LIN {X 0,Y 213.774,Z 837.959,A -85,B 0,C 180,E1 9874.512,E2 9874.512} C_VEL
LIN {X 0,Y 216.495,Z 837.046,A -85,B 0,C 180,E1 9873.088,E2 9873.088} C_VEL
LIN {X 0,Y 220.034,Z 835.344,A -85,B 0,C 180,E1 9871.796,E2 9871.796} C_VEL
LIN {X 0,Y 223.983,Z 833.719,A -85,B 0,C 180,E1 9870.296,E2 9870.296} C_VEL
LIN {X 0,Y 226.594,Z 832.46,A -85,B 0,C 180,E1 9869.505,E2 9869.505} C_VEL
LIN {X 0,Y 231.577,Z 830.349,A -85,B 0,C 180,E1 9867.921,E2 9867.921} C_VEL
LIN {X 0,Y 234.959,Z 828.778,A -85,B 0,C 180,E1 9866.995,E2 9866.995} C_VEL
LIN {X 0,Y 241.29,Z 825.829,A -85,B 0,C 180,E1 9865.408,E2 9865.408} C_VEL
LIN {X 0,Y 250.192,Z 821.605,A -85,B 0,C 180,E1 9863.446,E2 9863.446} C_VEL
LIN {X 0,Y 261.296,Z 816.099,A -85,B 0,C 180,E1 9861.41,E2 9861.41} C_VEL
LIN {X 0,Y 266.545,Z 813.328,A -85,B 0,C 180,E1 9860.587,E2 9860.587} C_VEL
LIN {X 0,Y 257.171,Z 829.628,A -85,B 0,C 180,E1 9857.623,E2 9857.623} C_VEL
LIN {X 0,Y 247.802,Z 844.317,A -85,B 0,C 180,E1 9854.272,E2 9854.272} C_VEL
LIN {X 0,Y 238.695,Z 857.461,A -85,B 0,C 180,E1 9850.488,E2 9850.488} C_VEL
LIN {X 0,Y 230.087,Z 869.099,A -85,B 0,C 180,E1 9846.229,E2 9846.229} C_VEL
LIN {X 0,Y 222.258,Z 879.206,A -85,B 0,C 180,E1 9841.457,E2 9841.457} C_VEL
LIN {X 0,Y 215.768,Z 887.387,A -85,B 0,C 180,E1 9836.415,E2 9836.415} C_VEL
LIN {X 0,Y 210.469,Z 894.092,A -85,B 0,C 180,E1 9830.874,E2 9830.874} C_VEL
LIN {X 0,Y 206.702,Z 899.028,A -85,B 0,C 180,E1 9825.143,E2 9825.143} C_VEL
LIN {X 0,Y 204.391,Z 902.303,A -85,B 0,C 180,E1 9819.291,E2 9819.291} C_VEL
LIN {X 0,Y 203.309,Z 903.961,A -85,B 0,C 180,E1 9813.384,E2 9813.384} C_VEL
LIN {X 0,Y 203.212,Z 904.09,A -85,B 0,C 180,E1 9807.744,E2 9807.744} C_VEL
LIN {X 0,Y 204.008,Z 902.842,A -85,B 0,C 180,E1 9802.112,E2 9802.112} C_VEL
LIN {X 0,Y 206.112,Z 899.833,A -85,B 0,C 180,E1 9795.963,E2 9795.963} C_VEL
LIN {X 0,Y 209.786,Z 895.013,A -85,B 0,C 180,E1 9789.93,E2 9789.93} C_VEL
LIN {X 0,Y 214.836,Z 888.617,A -85,B 0,C 180,E1 9784.352,E2 9784.352} C_VEL
LIN {X 0,Y 221.454,Z 880.322,A -85,B 0,C 180,E1 9779.021,E2 9779.021} C_VEL
LIN {X 0,Y 229.143,Z 870.475,A -85,B 0,C 180,E1 9774.217,E2 9774.217} C_VEL
LIN {X 0,Y 237.624,Z 859.12,A -85,B 0,C 180,E1 9769.924,E2 9769.924} C_VEL
LIN {X 0,Y 246.624,Z 846.271,A -85,B 0,C 180,E1 9766.109,E2 9766.109} C_VEL
LIN {X 0,Y 255.338,Z 832.826,A -85,B 0,C 180,E1 9762.922,E2 9762.922} C_VEL
LIN {X 0,Y 264.272,Z 817.707,A -85,B 0,C 180,E1 9760.032,E2 9760.032} C_VEL
LIN {X 0,Y 272.923,Z 801.409,A -85,B 0,C 180,E1 9757.517,E2 9757.517} C_VEL
LIN {X 0,Y 281.204,Z 783.726,A -85,B 0,C 180,E1 9755.309,E2 9755.309} C_VEL
LIN {X 0,Y 288.732,Z 765.064,A -85,B 0,C 180,E1 9753.427,E2 9753.427} C_VEL
LIN {X 0,Y 295.016,Z 746.597,A -85,B 0,C 180,E1 9751.92,E2 9751.92} C_VEL
LIN {X 0,Y 300.676,Z 726.186,A -85,B 0,C 180,E1 9750.584,E2 9750.584} C_VEL
LIN {X 0,Y 305.859,Z 701.959,A -85,B 0,C 180,E1 9749.35,E2 9749.35} C_VEL
LIN {X 0,Y 313.548,Z 662.516,A -85,B 0,C 180,E1 9747.755,E2 9747.755} C_VEL
LIN {X 0,Y 320.97,Z 622.102,A -85,B 0,C 180,E1 9746.524,E2 9746.524} C_VEL
LIN {X 0,Y 328.272,Z 576.098,A -85,B 0,C 180,E1 9745.404,E2 9745.404} C_VEL
LIN {X 0,Y 333.972,Z 529.706,A -85,B 0,C 180,E1 9744.467,E2 9744.467} C_VEL
LIN {X 0,Y 340.15,Z 466.539,A -85,B 0,C 180,E1 9743.356,E2 9743.356} C_VEL
LIN {X 0,Y 344.086,Z 450.132,A -85,B 0,C 180,E1 9742.901,E2 9742.901} C_VEL
LIN {X 0,Y 341.351,Z 438.925,A -85,B 0,C 180,E1 9739.82,E2 9739.82} C_VEL
LIN {X 0,Y 340.469,Z 435.442,A -85,B 0,C 180,E1 9738.706,E2 9738.706} C_VEL
LIN {X 0,Y 339.282,Z 432.899,A -85,B 0,C 180,E1 9737.488,E2 9737.488} C_VEL
LIN {X 0,Y 336.733,Z 431.213,A -85,B 0,C 180,E1 9735.367,E2 9735.367} C_VEL
LIN {X 0,Y 334.628,Z 429.482,A -85,B 0,C 180,E1 9733.301,E2 9733.301} C_VEL
LIN {X 0,Y 334.307,Z 428.715,A -85,B 0,C 180,E1 9732.841,E2 9732.841} C_VEL
LIN {X 0,Y 332.924,Z 422.507,A -85,B 0,C 180,E1 9729.421,E2 9729.421} C_VEL
LIN {X 0,Y 332.056,Z 418.778,A -85,B 0,C 180,E1 9726.571,E2 9726.571} C_VEL
LIN {X 0,Y 331.825,Z 415.306,A -85,B 0,C 180,E1 9722.936,E2 9722.936} C_VEL
LIN {X 0,Y 332.528,Z 414.439,A -85,B 0,C 180,E1 9717.932,E2 9717.932} C_VEL
LIN {X 0,Y 333.593,Z 415.275,A -85,B 0,C 180,E1 9715.186,E2 9715.186} C_VEL
LIN {X 0,Y 334.377,Z 429.017,A -85,B 0,C 180,E1 9710.621,E2 9710.621} C_VEL
LIN {X 0,Y 337.146,Z 447.925,A -85,B 0,C 180,E1 9705.443,E2 9705.443} C_VEL
LIN {X 0,Y 337.566,Z 450.515,A -85,B 0,C 180,E1 9704.861,E2 9704.861} C_VEL
LIN {X 0,Y 319.756,Z 552.113,A -85,B 0,C 180,E1 9702.274,E2 9702.274} C_VEL
LIN {X 0,Y 313.651,Z 616.805,A -85,B 0,C 180,E1 9700.912,E2 9700.912} C_VEL
LIN {X 0,Y 308.573,Z 653.152,A -85,B 0,C 180,E1 9700.066,E2 9700.066} C_VEL
LIN {X 0,Y 302.296,Z 687.872,A -85,B 0,C 180,E1 9699.032,E2 9699.032} C_VEL
LIN {X 0,Y 294.882,Z 721.646,A -85,B 0,C 180,E1 9697.789,E2 9697.789} C_VEL
LIN {X 0,Y 287.35,Z 751.978,A -85,B 0,C 180,E1 9696.384,E2 9696.384} C_VEL
LIN {X 0,Y 278.355,Z 784.046,A -85,B 0,C 180,E1 9694.465,E2 9694.465} C_VEL
LIN {X 0,Y 272.028,Z 802.983,A -85,B 0,C 180,E1 9693.044,E2 9693.044} C_VEL
LIN {X 0,Y 264.192,Z 822.641,A -85,B 0,C 180,E1 9691.182,E2 9691.182} C_VEL
LIN {X 0,Y 255.628,Z 841.24,A -85,B 0,C 180,E1 9688.939,E2 9688.939} C_VEL
LIN {X 0,Y 246.829,Z 858.228,A -85,B 0,C 180,E1 9686.353,E2 9686.353} C_VEL
LIN {X 0,Y 237.72,Z 874.11,A -85,B 0,C 180,E1 9683.325,E2 9683.325} C_VEL
LIN {X 0,Y 228.326,Z 889.305,A -85,B 0,C 180,E1 9679.639,E2 9679.639} C_VEL
LIN {X 0,Y 219.526,Z 902.891,A -85,B 0,C 180,E1 9675.457,E2 9675.457} C_VEL
LIN {X 0,Y 211.133,Z 915.618,A -85,B 0,C 180,E1 9670.452,E2 9670.452} C_VEL
LIN {X 0,Y 204.191,Z 926.472,A -85,B 0,C 180,E1 9664.955,E2 9664.955} C_VEL
LIN {X 0,Y 198.818,Z 935.674,A -85,B 0,C 180,E1 9658.868,E2 9658.868} C_VEL
LIN {X 0,Y 195.438,Z 942.931,A -85,B 0,C 180,E1 9652.564,E2 9652.564} C_VEL
LIN {X 0,Y 193.909,Z 948.606,A -85,B 0,C 180,E1 9645.86,E2 9645.86} C_VEL
LIN {X 0,Y 193.96,Z 952.104,A -85,B 0,C 180,E1 9639.795,E2 9639.795} C_VEL
LIN {X 0,Y 194.718,Z 953.916,A -85,B 0,C 180,E1 9634.417,E2 9634.417} C_VEL
LIN {X 0,Y 195.109,Z 954.446,A -85,B 0,C 180,E1 9630,E2 9630} C_VEL
LIN {X 0,Y 194.783,Z 953.918,A -85,B 0,C 180,E1 9625.584,E2 9625.584} C_VEL
LIN {X 0,Y 194.115,Z 952.266,A -85,B 0,C 180,E1 9619.913,E2 9619.913} C_VEL
LIN {X 0,Y 193.988,Z 951.89,A -85,B 0,C 180,E1 9613.223,E2 9613.223} C_VEL
LIN {X 0,Y 196.359,Z 949.933,A -85,B 0,C 180,E1 9605.319,E2 9605.319} C_VEL
LIN {X 0,Y 203.821,Z 945.545,A -85,B 0,C 180,E1 9595.996,E2 9595.996} C_VEL
LIN {X 0,Y 216.327,Z 939.485,A -85,B 0,C 180,E1 9587.559,E2 9587.559} C_VEL
LIN {X 0,Y 235.213,Z 931.168,A -85,B 0,C 180,E1 9579.697,E2 9579.697} C_VEL
LIN {X 0,Y 245.482,Z 926.927,A -85,B 0,C 180,E1 9576.57,E2 9576.57} C_VEL
LIN {X 0,Y 230.871,Z 927.562,A -85,B 0,C 180,E1 9571.896,E2 9571.896} C_VEL
LIN {X 0,Y 218.657,Z 926.56,A -85,B 0,C 180,E1 9566.625,E2 9566.625} C_VEL
LIN {X 0,Y 209.607,Z 924.018,A -85,B 0,C 180,E1 9561.257,E2 9561.257} C_VEL
LIN {X 0,Y 202.738,Z 919.727,A -85,B 0,C 180,E1 9555.446,E2 9555.446} C_VEL
LIN {X 0,Y 198.06,Z 913.469,A -85,B 0,C 180,E1 9549.297,E2 9549.297} C_VEL
LIN {X 0,Y 195.581,Z 905.888,A -85,B 0,C 180,E1 9543.517,E2 9543.517} C_VEL
LIN {X 0,Y 194.576,Z 897.367,A -85,B 0,C 180,E1 9538.233,E2 9538.233} C_VEL
LIN {X 0,Y 194.552,Z 887.031,A -85,B 0,C 180,E1 9532.915,E2 9532.915} C_VEL
LIN {X 0,Y 195.453,Z 874.895,A -85,B 0,C 180,E1 9527.718,E2 9527.718} C_VEL
LIN {X 0,Y 197.218,Z 861.476,A -85,B 0,C 180,E1 9522.899,E2 9522.899} C_VEL
LIN {X 0,Y 199.677,Z 847.469,A -85,B 0,C 180,E1 9518.558,E2 9518.558} C_VEL
LIN {X 0,Y 201.324,Z 847.012,A -85,B 0,C 180,E1 9517.208,E2 9517.208} C_VEL
LIN {X 0,Y 204.017,Z 845.607,A -85,B 0,C 180,E1 9515.997,E2 9515.997} C_VEL
LIN {X 0,Y 206.542,Z 844.763,A -85,B 0,C 180,E1 9514.478,E2 9514.478} C_VEL
LIN {X 0,Y 209.844,Z 843.247,A -85,B 0,C 180,E1 9513.085,E2 9513.085} C_VEL
LIN {X 0,Y 213.572,Z 841.761,A -85,B 0,C 180,E1 9511.475,E2 9511.475} C_VEL
LIN {X 0,Y 215.992,Z 840.669,A -85,B 0,C 180,E1 9510.613,E2 9510.613} C_VEL
LIN {X 0,Y 220.769,Z 838.719,A -85,B 0,C 180,E1 9508.914,E2 9508.914} C_VEL
LIN {X 0,Y 229.354,Z 835.015,A -85,B 0,C 180,E1 9506.376,E2 9506.376} C_VEL
LIN {X 0,Y 237.845,Z 831.343,A -85,B 0,C 180,E1 9504.243,E2 9504.243} C_VEL
LIN {X 0,Y 247.768,Z 826.829,A -85,B 0,C 180,E1 9502.163,E2 9502.163} C_VEL
LIN {X 0,Y 256.771,Z 822.752,A -85,B 0,C 180,E1 9500.496,E2 9500.496} C_VEL
LIN {X 0,Y 247.225,Z 837.953,A -85,B 0,C 180,E1 9497.4,E2 9497.4} C_VEL
LIN {X 0,Y 237.316,Z 852.257,A -85,B 0,C 180,E1 9493.709,E2 9493.709} C_VEL
LIN {X 0,Y 228.297,Z 864.319,A -85,B 0,C 180,E1 9489.751,E2 9489.751} C_VEL
LIN {X 0,Y 219.841,Z 874.97,A -85,B 0,C 180,E1 9485.284,E2 9485.284} C_VEL
LIN {X 0,Y 212.23,Z 884.171,A -85,B 0,C 180,E1 9480.273,E2 9480.273} C_VEL
LIN {X 0,Y 205.696,Z 891.933,A -85,B 0,C 180,E1 9474.631,E2 9474.631} C_VEL
LIN {X 0,Y 200.728,Z 897.907,A -85,B 0,C 180,E1 9468.591,E2 9468.591} C_VEL
LIN {X 0,Y 197.535,Z 901.951,A -85,B 0,C 180,E1 9462.572,E2 9462.572} C_VEL
LIN {X 0,Y 195.79,Z 904.377,A -85,B 0,C 180,E1 9456.451,E2 9456.451} C_VEL
LIN {X 0,Y 195.217,Z 905.198,A -85,B 0,C 180,E1 9450.587,E2 9450.587} C_VEL
LIN {X 0,Y 195.576,Z 904.642,A -85,B 0,C 180,E1 9444.72,E2 9444.72} C_VEL
LIN {X 0,Y 197.067,Z 902.567,A -85,B 0,C 180,E1 9438.587,E2 9438.587} C_VEL
LIN {X 0,Y 200.126,Z 898.677,A -85,B 0,C 180,E1 9432.256,E2 9432.256} C_VEL
LIN {X 0,Y 204.905,Z 892.926,A -85,B 0,C 180,E1 9426.108,E2 9426.108} C_VEL
LIN {X 0,Y 211.121,Z 885.568,A -85,B 0,C 180,E1 9420.492,E2 9420.492} C_VEL
LIN {X 0,Y 218.51,Z 876.704,A -85,B 0,C 180,E1 9415.43,E2 9415.43} C_VEL
LIN {X 0,Y 226.846,Z 866.319,A -85,B 0,C 180,E1 9410.876,E2 9410.876} C_VEL
LIN {X 0,Y 235.805,Z 854.497,A -85,B 0,C 180,E1 9406.831,E2 9406.831} C_VEL
LIN {X 0,Y 245.117,Z 841.277,A -85,B 0,C 180,E1 9403.26,E2 9403.26} C_VEL
LIN {X 0,Y 254.736,Z 826.348,A -85,B 0,C 180,E1 9400.056,E2 9400.056} C_VEL
LIN {X 0,Y 264.011,Z 810.344,A -85,B 0,C 180,E1 9397.313,E2 9397.313} C_VEL
LIN {X 0,Y 272.725,Z 793.383,A -85,B 0,C 180,E1 9394.974,E2 9394.974} C_VEL
LIN {X 0,Y 280.716,Z 775.526,A -85,B 0,C 180,E1 9392.983,E2 9392.983} C_VEL
LIN {X 0,Y 287.85,Z 756.807,A -85,B 0,C 180,E1 9391.294,E2 9391.294} C_VEL
LIN {X 0,Y 294.047,Z 737.187,A -85,B 0,C 180,E1 9389.875,E2 9389.875} C_VEL
LIN {X 0,Y 299.024,Z 717.296,A -85,B 0,C 180,E1 9388.727,E2 9388.727} C_VEL
LIN {X 0,Y 306.803,Z 679.572,A -85,B 0,C 180,E1 9387.046,E2 9387.046} C_VEL
LIN {X 0,Y 314.484,Z 640.094,A -85,B 0,C 180,E1 9385.7,E2 9385.7} C_VEL
LIN {X 0,Y 322.291,Z 594.861,A -85,B 0,C 180,E1 9384.537,E2 9384.537} C_VEL
LIN {X 0,Y 328.535,Z 550.082,A -85,B 0,C 180,E1 9383.578,E2 9383.578} C_VEL
LIN {X 0,Y 334.258,Z 494.763,A -85,B 0,C 180,E1 9382.586,E2 9382.586} C_VEL
LIN {X 0,Y 336.896,Z 469.242,A -85,B 0,C 180,E1 9382.144,E2 9382.144} C_VEL
LIN {X 0,Y 340.426,Z 454.288,A -85,B 0,C 180,E1 9381.721,E2 9381.721} C_VEL
LIN {X 0,Y 338.052,Z 443.9,A -85,B 0,C 180,E1 9378.719,E2 9378.719} C_VEL
LIN {X 0,Y 335.855,Z 434.787,A -85,B 0,C 180,E1 9375.498,E2 9375.498} C_VEL
LIN {X 0,Y 334.307,Z 428.715,A -85,B 0,C 180,E1 9372.841,E2 9372.841} C_VEL
LIN {X 0,Y 333.429,Z 427.235,A -85,B 0,C 180,E1 9371.542,E2 9371.542} C_VEL
LIN {X 0,Y 331.509,Z 427.281,A -85,B 0,C 180,E1 9369.153,E2 9369.153} C_VEL
LIN {X 0,Y 330.247,Z 427.072,A -85,B 0,C 180,E1 9367.119,E2 9367.119} C_VEL
LIN {X 0,Y 330.126,Z 426.75,A -85,B 0,C 180,E1 9366.734,E2 9366.734} C_VEL
LIN {X 0,Y 329.901,Z 423.004,A -85,B 0,C 180,E1 9362.606,E2 9362.606} C_VEL
LIN {X 0,Y 330.781,Z 422.255,A -85,B 0,C 180,E1 9357.748,E2 9357.748} C_VEL
LIN {X 0,Y 331.614,Z 422.963,A -85,B 0,C 180,E1 9355.504,E2 9355.504} C_VEL
LIN {X 0,Y 332.18,Z 436.644,A -85,B 0,C 180,E1 9350.995,E2 9350.995} C_VEL
LIN {X 0,Y 334.634,Z 454.529,A -85,B 0,C 180,E1 9346.085,E2 9346.085} C_VEL
LIN {X 0,Y 317.576,Z 549.187,A -85,B 0,C 180,E1 9343.709,E2 9343.709} C_VEL
LIN {X 0,Y 311.251,Z 614.325,A -85,B 0,C 180,E1 9342.345,E2 9342.345} C_VEL
LIN {X 0,Y 305.933,Z 651.501,A -85,B 0,C 180,E1 9341.503,E2 9341.503} C_VEL
LIN {X 0,Y 299.223,Z 687.667,A -85,B 0,C 180,E1 9340.448,E2 9340.448} C_VEL
LIN {X 0,Y 291.638,Z 721.28,A -85,B 0,C 180,E1 9339.23,E2 9339.23} C_VEL
LIN {X 0,Y 283.713,Z 752.096,A -85,B 0,C 180,E1 9337.821,E2 9337.821} C_VEL
LIN {X 0,Y 275.126,Z 782.04,A -85,B 0,C 180,E1 9336.064,E2 9336.064} C_VEL
LIN {X 0,Y 268.417,Z 801.547,A -85,B 0,C 180,E1 9334.634,E2 9334.634} C_VEL
LIN {X 0,Y 260.644,Z 820.526,A -85,B 0,C 180,E1 9332.874,E2 9332.874} C_VEL
LIN {X 0,Y 252.122,Z 838.586,A -85,B 0,C 180,E1 9330.75,E2 9330.75} C_VEL
LIN {X 0,Y 243.257,Z 855.197,A -85,B 0,C 180,E1 9328.305,E2 9328.305} C_VEL
LIN {X 0,Y 233.594,Z 871.554,A -85,B 0,C 180,E1 9325.27,E2 9325.27} C_VEL
LIN {X 0,Y 224.091,Z 886.437,A -85,B 0,C 180,E1 9321.749,E2 9321.749} C_VEL
LIN {X 0,Y 214.948,Z 899.902,A -85,B 0,C 180,E1 9317.7,E2 9317.7} C_VEL
LIN {X 0,Y 206.322,Z 912.249,A -85,B 0,C 180,E1 9312.963,E2 9312.963} C_VEL
LIN {X 0,Y 198.346,Z 923.808,A -85,B 0,C 180,E1 9307.224,E2 9307.224} C_VEL
LIN {X 0,Y 192.471,Z 932.966,A -85,B 0,C 180,E1 9301.299,E2 9301.299} C_VEL
LIN {X 0,Y 188.332,Z 940.658,A -85,B 0,C 180,E1 9294.787,E2 9294.787} C_VEL
LIN {X 0,Y 186.215,Z 946.456,A -85,B 0,C 180,E1 9288.118,E2 9288.118} C_VEL
LIN {X 0,Y 185.881,Z 950.495,A -85,B 0,C 180,E1 9281.48,E2 9281.48} C_VEL
LIN {X 0,Y 186.572,Z 952.702,A -85,B 0,C 180,E1 9275.536,E2 9275.536} C_VEL
LIN {X 0,Y 187.122,Z 953.372,A -85,B 0,C 180,E1 9271.225,E2 9271.225} C_VEL
LIN {X 0,Y 187.016,Z 953.251,A -85,B 0,C 180,E1 9267.242,E2 9267.242} C_VEL
LIN {X 0,Y 186.372,Z 951.942,A -85,B 0,C 180,E1 9261.981,E2 9261.981} C_VEL
LIN {X 0,Y 186.121,Z 950.581,A -85,B 0,C 180,E1 9258.22,E2 9258.22} C_VEL
LIN {X 0,Y 186.54,Z 950.022,A -85,B 0,C 180,E1 9250.589,E2 9250.589} C_VEL
LIN {X 0,Y 190.211,Z 947.854,A -85,B 0,C 180,E1 9242.105,E2 9242.105} C_VEL
LIN {X 0,Y 200.211,Z 943.1,A -85,B 0,C 180,E1 9232.1,E2 9232.1} C_VEL
LIN {X 0,Y 215.395,Z 936.848,A -85,B 0,C 180,E1 9223.6,E2 9223.6} C_VEL
LIN {X 0,Y 235.218,Z 929.227,A -85,B 0,C 180,E1 9216.522,E2 9216.522} C_VEL
LIN {X 0,Y 220.878,Z 928.989,A -85,B 0,C 180,E1 9211.676,E2 9211.676} C_VEL
LIN {X 0,Y 208.835,Z 927.095,A -85,B 0,C 180,E1 9206.135,E2 9206.135} C_VEL
LIN {X 0,Y 200.03,Z 923.715,A -85,B 0,C 180,E1 9200.482,E2 9200.482} C_VEL
LIN {X 0,Y 193.497,Z 918.5,A -85,B 0,C 180,E1 9194.362,E2 9194.362} C_VEL
LIN {X 0,Y 189.37,Z 911.663,A -85,B 0,C 180,E1 9188.196,E2 9188.196} C_VEL
LIN {X 0,Y 187.278,Z 903.762,A -85,B 0,C 180,E1 9182.448,E2 9182.448} C_VEL
LIN {X 0,Y 186.475,Z 894.015,A -85,B 0,C 180,E1 9176.619,E2 9176.619} C_VEL
LIN {X 0,Y 186.765,Z 882.809,A -85,B 0,C 180,E1 9171.068,E2 9171.068} C_VEL
LIN {X 0,Y 187.99,Z 870.181,A -85,B 0,C 180,E1 9165.838,E2 9165.838} C_VEL
LIN {X 0,Y 190.271,Z 855.222,A -85,B 0,C 180,E1 9160.666,E2 9160.666} C_VEL
LIN {X 0,Y 190.434,Z 854.584,A -85,B 0,C 180,E1 9160.364,E2 9160.364} C_VEL
LIN {X 0,Y 191.918,Z 854.122,A -85,B 0,C 180,E1 9158.931,E2 9158.931} C_VEL
LIN {X 0,Y 194.691,Z 852.79,A -85,B 0,C 180,E1 9157.345,E2 9157.345} C_VEL
LIN {X 0,Y 197.716,Z 851.58,A -85,B 0,C 180,E1 9155.5,E2 9155.5} C_VEL
LIN {X 0,Y 199.738,Z 850.686,A -85,B 0,C 180,E1 9154.5,E2 9154.5} C_VEL
LIN {X 0,Y 203.867,Z 849.004,A -85,B 0,C 180,E1 9152.546,E2 9152.546} C_VEL
LIN {X 0,Y 210.165,Z 846.505,A -85,B 0,C 180,E1 9149.985,E2 9149.985} C_VEL
LIN {X 0,Y 217.554,Z 843.54,A -85,B 0,C 180,E1 9147.47,E2 9147.47} C_VEL
LIN {X 0,Y 225.682,Z 840.264,A -85,B 0,C 180,E1 9145.142,E2 9145.142} C_VEL
LIN {X 0,Y 235.195,Z 836.31,A -85,B 0,C 180,E1 9142.865,E2 9142.865} C_VEL
LIN {X 0,Y 246.225,Z 831.487,A -85,B 0,C 180,E1 9140.691,E2 9140.691} C_VEL
LIN {X 0,Y 247.205,Z 831.074,A -85,B 0,C 180,E1 9140.502,E2 9140.502} C_VEL
LIN {X 0,Y 237.234,Z 845.705,A -85,B 0,C 180,E1 9137.17,E2 9137.17} C_VEL
LIN {X 0,Y 227.334,Z 858.969,A -85,B 0,C 180,E1 9133.326,E2 9133.326} C_VEL
LIN {X 0,Y 217.886,Z 870.69,A -85,B 0,C 180,E1 9128.955,E2 9128.955} C_VEL
LIN {X 0,Y 209.2,Z 880.866,A -85,B 0,C 180,E1 9124.002,E2 9124.002} C_VEL
LIN {X 0,Y 201.59,Z 889.464,A -85,B 0,C 180,E1 9118.435,E2 9118.435} C_VEL
LIN {X 0,Y 195.631,Z 896.147,A -85,B 0,C 180,E1 9112.541,E2 9112.541} C_VEL
LIN {X 0,Y 191.358,Z 901.064,A -85,B 0,C 180,E1 9106.39,E2 9106.39} C_VEL
LIN {X 0,Y 188.707,Z 904.318,A -85,B 0,C 180,E1 9100.07,E2 9100.07} C_VEL
LIN {X 0,Y 187.458,Z 905.963,A -85,B 0,C 180,E1 9093.67,E2 9093.67} C_VEL
LIN {X 0,Y 187.348,Z 906.093,A -85,B 0,C 180,E1 9087.553,E2 9087.553} C_VEL
LIN {X 0,Y 188.268,Z 904.854,A -85,B 0,C 180,E1 9081.448,E2 9081.448} C_VEL
LIN {X 0,Y 190.688,Z 901.864,A -85,B 0,C 180,E1 9074.801,E2 9074.801} C_VEL
LIN {X 0,Y 194.864,Z 897.067,A -85,B 0,C 180,E1 9068.319,E2 9068.319} C_VEL
LIN {X 0,Y 200.552,Z 890.69,A -85,B 0,C 180,E1 9062.376,E2 9062.376} C_VEL
LIN {X 0,Y 207.917,Z 882.411,A -85,B 0,C 180,E1 9056.754,E2 9056.754} C_VEL
LIN {X 0,Y 216.245,Z 872.748,A -85,B 0,C 180,E1 9051.819,E2 9051.819} C_VEL
LIN {X 0,Y 225.396,Z 861.565,A -85,B 0,C 180,E1 9047.426,E2 9047.426} C_VEL
LIN {X 0,Y 234.952,Z 849.037,A -85,B 0,C 180,E1 9043.585,E2 9043.585} C_VEL
LIN {X 0,Y 244.778,Z 835.009,A -85,B 0,C 180,E1 9040.193,E2 9040.193} C_VEL
LIN {X 0,Y 254.613,Z 819.47,A -85,B 0,C 180,E1 9037.213,E2 9037.213} C_VEL
LIN {X 0,Y 263.892,Z 803.012,A -85,B 0,C 180,E1 9034.693,E2 9034.693} C_VEL
LIN {X 0,Y 272.434,Z 785.735,A -85,B 0,C 180,E1 9032.563,E2 9032.563} C_VEL
LIN {X 0,Y 279.957,Z 768.107,A -85,B 0,C 180,E1 9030.799,E2 9030.799} C_VEL
LIN {X 0,Y 286.635,Z 749.617,A -85,B 0,C 180,E1 9029.297,E2 9029.297} C_VEL
LIN {X 0,Y 292.294,Z 730.504,A -85,B 0,C 180,E1 9028.046,E2 9028.046} C_VEL
LIN {X 0,Y 297.469,Z 708.123,A -85,B 0,C 180,E1 9026.886,E2 9026.886} C_VEL
LIN {X 0,Y 305.494,Z 669.757,A -85,B 0,C 180,E1 9025.302,E2 9025.302} C_VEL
LIN {X 0,Y 313.232,Z 629.98,A -85,B 0,C 180,E1 9024.068,E2 9024.068} C_VEL
LIN {X 0,Y 320.771,Z 585.376,A -85,B 0,C 180,E1 9022.996,E2 9022.996} C_VEL
LIN {X 0,Y 326.845,Z 539.857,A -85,B 0,C 180,E1 9022.078,E2 9022.078} C_VEL
LIN {X 0,Y 333.775,Z 472.082,A -85,B 0,C 180,E1 9020.911,E2 9020.911} C_VEL
LIN {X 0,Y 336.956,Z 458.646,A -85,B 0,C 180,E1 9020.543,E2 9020.543} C_VEL
LIN {X 0,Y 334.834,Z 448.807,A -85,B 0,C 180,E1 9017.554,E2 9017.554} C_VEL
LIN {X 0,Y 333.061,Z 440.864,A -85,B 0,C 180,E1 9014.607,E2 9014.607} C_VEL
LIN {X 0,Y 331.576,Z 434.33,A -85,B 0,C 180,E1 9011.568,E2 9011.568} C_VEL
LIN {X 0,Y 330.555,Z 429.261,A -85,B 0,C 180,E1 9008.524,E2 9008.524} C_VEL
LIN {X 0,Y 330.126,Z 426.75,A -85,B 0,C 180,E1 9006.734,E2 9006.734} C_VEL
LIN {X 0,Y 329.666,Z 426.429,A -85,B 0,C 180,E1 9005.386,E2 9005.386} C_VEL
LIN {X 0,Y 328.616,Z 428.738,A -85,B 0,C 180,E1 9002.979,E2 9002.979} C_VEL
LIN {X 0,Y 328.152,Z 430.31,A -85,B 0,C 180,E1 9001.029,E2 9001.029} C_VEL
LIN {X 0,Y 328.183,Z 430.311,A -85,B 0,C 180,E1 9000.537,E2 9000.537} C_VEL
LIN {X 0,Y 329.15,Z 430.15,A -85,B 0,C 180,E1 8997.04,E2 8997.04} C_VEL
LIN {X 0,Y 329.646,Z 430.754,A -85,B 0,C 180,E1 8995.782,E2 8995.782} C_VEL
LIN {X 0,Y 330.058,Z 443.709,A -85,B 0,C 180,E1 8991.551,E2 8991.551} C_VEL
LIN {X 0,Y 331.816,Z 458.871,A -85,B 0,C 180,E1 8987.325,E2 8987.325} C_VEL
LIN {X 0,Y 315.61,Z 546.131,A -85,B 0,C 180,E1 8985.166,E2 8985.166} C_VEL
LIN {X 0,Y 309.065,Z 611.623,A -85,B 0,C 180,E1 8983.812,E2 8983.812} C_VEL
LIN {X 0,Y 303.553,Z 649.408,A -85,B 0,C 180,E1 8982.974,E2 8982.974} C_VEL
LIN {X 0,Y 296.75,Z 685.329,A -85,B 0,C 180,E1 8981.957,E2 8981.957} C_VEL
LIN {X 0,Y 289.056,Z 718.97,A -85,B 0,C 180,E1 8980.777,E2 8980.777} C_VEL
LIN {X 0,Y 280.917,Z 750.037,A -85,B 0,C 180,E1 8979.409,E2 8979.409} C_VEL
LIN {X 0,Y 271.892,Z 780.773,A -85,B 0,C 180,E1 8977.653,E2 8977.653} C_VEL
LIN {X 0,Y 264.922,Z 800.426,A -85,B 0,C 180,E1 8976.243,E2 8976.243} C_VEL
LIN {X 0,Y 256.966,Z 819.279,A -85,B 0,C 180,E1 8974.521,E2 8974.521} C_VEL
LIN {X 0,Y 248.159,Z 837.343,A -85,B 0,C 180,E1 8972.428,E2 8972.428} C_VEL
LIN {X 0,Y 238.952,Z 853.946,A -85,B 0,C 180,E1 8970.019,E2 8970.019} C_VEL
LIN {X 0,Y 228.906,Z 870.34,A -85,B 0,C 180,E1 8967.001,E2 8967.001} C_VEL
LIN {X 0,Y 218.97,Z 885.214,A -85,B 0,C 180,E1 8963.482,E2 8963.482} C_VEL
LIN {X 0,Y 209.353,Z 898.701,A -85,B 0,C 180,E1 8959.411,E2 8959.411} C_VEL
LIN {X 0,Y 200.403,Z 910.85,A -85,B 0,C 180,E1 8954.709,E2 8954.709} C_VEL
LIN {X 0,Y 192.068,Z 922.146,A -85,B 0,C 180,E1 8949.044,E2 8949.044} C_VEL
LIN {X 0,Y 185.619,Z 931.433,A -85,B 0,C 180,E1 8942.961,E2 8942.961} C_VEL
LIN {X 0,Y 180.96,Z 939.232,A -85,B 0,C 180,E1 8936.234,E2 8936.234} C_VEL
LIN {X 0,Y 178.449,Z 945.149,A -85,B 0,C 180,E1 8929.304,E2 8929.304} C_VEL
LIN {X 0,Y 177.881,Z 949.309,A -85,B 0,C 180,E1 8922.333,E2 8922.333} C_VEL
LIN {X 0,Y 178.527,Z 951.616,A -85,B 0,C 180,E1 8916.108,E2 8916.108} C_VEL
LIN {X 0,Y 179.15,Z 952.346,A -85,B 0,C 180,E1 8911.599,E2 8911.599} C_VEL
LIN {X 0,Y 179.119,Z 952.298,A -85,B 0,C 180,E1 8907.752,E2 8907.752} C_VEL
LIN {X 0,Y 178.478,Z 951.231,A -85,B 0,C 180,E1 8902.575,E2 8902.575} C_VEL
LIN {X 0,Y 178.201,Z 948.82,A -85,B 0,C 180,E1 8896.099,E2 8896.099} C_VEL
LIN {X 0,Y 179.565,Z 948.028,A -85,B 0,C 180,E1 8887.404,E2 8887.404} C_VEL
LIN {X 0,Y 184.909,Z 945.615,A -85,B 0,C 180,E1 8878.363,E2 8878.363} C_VEL
LIN {X 0,Y 198.035,Z 940.497,A -85,B 0,C 180,E1 8867.815,E2 8867.815} C_VEL
LIN {X 0,Y 215.595,Z 934.277,A -85,B 0,C 180,E1 8859.657,E2 8859.657} C_VEL
LIN {X 0,Y 224.946,Z 931.062,A -85,B 0,C 180,E1 8856.479,E2 8856.479} C_VEL
LIN {X 0,Y 210.323,Z 929.897,A -85,B 0,C 180,E1 8851.211,E2 8851.211} C_VEL
LIN {X 0,Y 199.011,Z 927.195,A -85,B 0,C 180,E1 8845.6,E2 8845.6} C_VEL
LIN {X 0,Y 190.144,Z 922.711,A -85,B 0,C 180,E1 8839.347,E2 8839.347} C_VEL
LIN {X 0,Y 184.091,Z 916.502,A -85,B 0,C 180,E1 8832.867,E2 8832.867} C_VEL
LIN {X 0,Y 180.604,Z 909.093,A -85,B 0,C 180,E1 8826.677,E2 8826.677} C_VEL
LIN {X 0,Y 178.898,Z 900.333,A -85,B 0,C 180,E1 8820.64,E2 8820.64} C_VEL
LIN {X 0,Y 178.467,Z 890.241,A -85,B 0,C 180,E1 8814.857,E2 8814.857} C_VEL
LIN {X 0,Y 179.045,Z 878.857,A -85,B 0,C 180,E1 8809.38,E2 8809.38} C_VEL
LIN {X 0,Y 180.645,Z 865.331,A -85,B 0,C 180,E1 8803.933,E2 8803.933} C_VEL
LIN {X 0,Y 181.259,Z 861.357,A -85,B 0,C 180,E1 8802.504,E2 8802.504} C_VEL
LIN {X 0,Y 182.655,Z 860.881,A -85,B 0,C 180,E1 8800.825,E2 8800.825} C_VEL
LIN {X 0,Y 184.878,Z 859.719,A -85,B 0,C 180,E1 8799.418,E2 8799.418} C_VEL
LIN {X 0,Y 187.455,Z 858.737,A -85,B 0,C 180,E1 8797.415,E2 8797.415} C_VEL
LIN {X 0,Y 189.402,Z 857.837,A -85,B 0,C 180,E1 8796.345,E2 8796.345} C_VEL
LIN {X 0,Y 193.084,Z 856.41,A -85,B 0,C 180,E1 8794.215,E2 8794.215} C_VEL
LIN {X 0,Y 199.5,Z 853.891,A -85,B 0,C 180,E1 8791.239,E2 8791.239} C_VEL
LIN {X 0,Y 205.998,Z 851.449,A -85,B 0,C 180,E1 8788.681,E2 8788.681} C_VEL
LIN {X 0,Y 213.66,Z 848.533,A -85,B 0,C 180,E1 8786.158,E2 8786.158} C_VEL
LIN {X 0,Y 222.793,Z 845.011,A -85,B 0,C 180,E1 8783.671,E2 8783.671} C_VEL
LIN {X 0,Y 232.579,Z 841.124,A -85,B 0,C 180,E1 8781.437,E2 8781.437} C_VEL
LIN {X 0,Y 237.354,Z 839.232,A -85,B 0,C 180,E1 8780.437,E2 8780.437} C_VEL
LIN {X 0,Y 227.209,Z 852.939,A -85,B 0,C 180,E1 8776.931,E2 8776.931} C_VEL
LIN {X 0,Y 217.313,Z 865.212,A -85,B 0,C 180,E1 8772.92,E2 8772.92} C_VEL
LIN {X 0,Y 207.93,Z 876.049,A -85,B 0,C 180,E1 8768.341,E2 8768.341} C_VEL
LIN {X 0,Y 199.311,Z 885.495,A -85,B 0,C 180,E1 8763.092,E2 8763.092} C_VEL
LIN {X 0,Y 191.988,Z 893.271,A -85,B 0,C 180,E1 8757.278,E2 8757.278} C_VEL
LIN {X 0,Y 186.123,Z 899.5,A -85,B 0,C 180,E1 8750.767,E2 8750.767} C_VEL
LIN {X 0,Y 182.16,Z 903.835,A -85,B 0,C 180,E1 8743.976,E2 8743.976} C_VEL
LIN {X 0,Y 180.068,Z 906.292,A -85,B 0,C 180,E1 8737.338,E2 8737.338} C_VEL
LIN {X 0,Y 179.346,Z 907.18,A -85,B 0,C 180,E1 8730.959,E2 8730.959} C_VEL
LIN {X 0,Y 179.713,Z 906.706,A -85,B 0,C 180,E1 8724.573,E2 8724.573} C_VEL
LIN {X 0,Y 181.37,Z 904.722,A -85,B 0,C 180,E1 8717.908,E2 8717.908} C_VEL
LIN {X 0,Y 184.599,Z 901.148,A -85,B 0,C 180,E1 8711.363,E2 8711.363} C_VEL
LIN {X 0,Y 189.559,Z 895.888,A -85,B 0,C 180,E1 8705.04,E2 8705.04} C_VEL
LIN {X 0,Y 195.918,Z 889.209,A -85,B 0,C 180,E1 8699.312,E2 8699.312} C_VEL
LIN {X 0,Y 203.809,Z 880.749,A -85,B 0,C 180,E1 8693.934,E2 8693.934} C_VEL
LIN {X 0,Y 212.618,Z 870.897,A -85,B 0,C 180,E1 8689.18,E2 8689.18} C_VEL
LIN {X 0,Y 222.139,Z 859.575,A -85,B 0,C 180,E1 8684.966,E2 8684.966} C_VEL
LIN {X 0,Y 232.373,Z 846.387,A -85,B 0,C 180,E1 8681.148,E2 8681.148} C_VEL
LIN {X 0,Y 242.393,Z 832.229,A -85,B 0,C 180,E1 8677.926,E2 8677.926} C_VEL
LIN {X 0,Y 252.019,Z 817.122,A -85,B 0,C 180,E1 8675.184,E2 8675.184} C_VEL
LIN {X 0,Y 261.527,Z 800.292,A -85,B 0,C 180,E1 8672.741,E2 8672.741} C_VEL
LIN {X 0,Y 270.277,Z 782.497,A -85,B 0,C 180,E1 8670.669,E2 8670.669} C_VEL
LIN {X 0,Y 277.78,Z 764.721,A -85,B 0,C 180,E1 8668.991,E2 8668.991} C_VEL
LIN {X 0,Y 284.302,Z 746.388,A -85,B 0,C 180,E1 8667.59,E2 8667.59} C_VEL
LIN {X 0,Y 290.104,Z 726.061,A -85,B 0,C 180,E1 8666.346,E2 8666.346} C_VEL
LIN {X 0,Y 298.349,Z 689.251,A -85,B 0,C 180,E1 8664.637,E2 8664.637} C_VEL
LIN {X 0,Y 306.571,Z 649.532,A -85,B 0,C 180,E1 8663.237,E2 8663.237} C_VEL
LIN {X 0,Y 314.849,Z 604.958,A -85,B 0,C 180,E1 8662.084,E2 8662.084} C_VEL
LIN {X 0,Y 321.643,Z 559.447,A -85,B 0,C 180,E1 8661.121,E2 8661.121} C_VEL
LIN {X 0,Y 326.935,Z 512.22,A -85,B 0,C 180,E1 8660.28,E2 8660.28} C_VEL
LIN {X 0,Y 330.832,Z 474.84,A -85,B 0,C 180,E1 8659.653,E2 8659.653} C_VEL
LIN {X 0,Y 333.615,Z 463.08,A -85,B 0,C 180,E1 8659.341,E2 8659.341} C_VEL
LIN {X 0,Y 331.652,Z 453.139,A -85,B 0,C 180,E1 8656.148,E2 8656.148} C_VEL
LIN {X 0,Y 330.07,Z 445.457,A -85,B 0,C 180,E1 8653.043,E2 8653.043} C_VEL
LIN {X 0,Y 328.824,Z 439.214,A -85,B 0,C 180,E1 8649.804,E2 8649.804} C_VEL
LIN {X 0,Y 328.084,Z 434.344,A -85,B 0,C 180,E1 8646.475,E2 8646.475} C_VEL
LIN {X 0,Y 328.08,Z 430.764,A -85,B 0,C 180,E1 8642.445,E2 8642.445} C_VEL
LIN {X 0,Y 328.183,Z 430.311,A -85,B 0,C 180,E1 8640.537,E2 8640.537} C_VEL
LIN {X 0,Y 328.234,Z 430.925,A -85,B 0,C 180,E1 8639.278,E2 8639.278} C_VEL
LIN {X 0,Y 328.04,Z 433.786,A -85,B 0,C 180,E1 8637.693,E2 8637.693} C_VEL
LIN {X 0,Y 327.611,Z 441.652,A -85,B 0,C 180,E1 8635.019,E2 8635.019} C_VEL
LIN {X 0,Y 327.603,Z 442.751,A -85,B 0,C 180,E1 8634.666,E2 8634.666} C_VEL
LIN {X 0,Y 327.955,Z 451.516,A -85,B 0,C 180,E1 8631.894,E2 8631.894} C_VEL
LIN {X 0,Y 329.07,Z 463.463,A -85,B 0,C 180,E1 8628.567,E2 8628.567} C_VEL
LIN {X 0,Y 313.808,Z 543.454,A -85,B 0,C 180,E1 8626.635,E2 8626.635} C_VEL
LIN {X 0,Y 307.081,Z 608.92,A -85,B 0,C 180,E1 8625.3,E2 8625.3} C_VEL
LIN {X 0,Y 301.411,Z 647.092,A -85,B 0,C 180,E1 8624.472,E2 8624.472} C_VEL
LIN {X 0,Y 294.353,Z 683.739,A -85,B 0,C 180,E1 8623.468,E2 8623.468} C_VEL
LIN {X 0,Y 286.597,Z 716.892,A -85,B 0,C 180,E1 8622.343,E2 8622.343} C_VEL
LIN {X 0,Y 278.138,Z 748.638,A -85,B 0,C 180,E1 8620.991,E2 8620.991} C_VEL
LIN {X 0,Y 268.869,Z 779.544,A -85,B 0,C 180,E1 8619.276,E2 8619.276} C_VEL
LIN {X 0,Y 261.589,Z 799.487,A -85,B 0,C 180,E1 8617.879,E2 8617.879} C_VEL
LIN {X 0,Y 253.148,Z 818.845,A -85,B 0,C 180,E1 8616.135,E2 8616.135} C_VEL
LIN {X 0,Y 244.04,Z 836.835,A -85,B 0,C 180,E1 8614.072,E2 8614.072} C_VEL
LIN {X 0,Y 234.164,Z 853.928,A -85,B 0,C 180,E1 8611.597,E2 8611.597} C_VEL
LIN {X 0,Y 223.428,Z 870.565,A -85,B 0,C 180,E1 8608.488,E2 8608.488} C_VEL
LIN {X 0,Y 212.82,Z 885.678,A -85,B 0,C 180,E1 8604.835,E2 8604.835} C_VEL
LIN {X 0,Y 202.292,Z 899.686,A -85,B 0,C 180,E1 8600.45,E2 8600.45} C_VEL
LIN {X 0,Y 192.565,Z 912.154,A -85,B 0,C 180,E1 8595.346,E2 8595.346} C_VEL
LIN {X 0,Y 184.042,Z 923.07,A -85,B 0,C 180,E1 8589.468,E2 8589.468} C_VEL
LIN {X 0,Y 177.196,Z 932.344,A -85,B 0,C 180,E1 8582.8,E2 8582.8} C_VEL
LIN {X 0,Y 172.463,Z 939.992,A -85,B 0,C 180,E1 8575.406,E2 8575.406} C_VEL
LIN {X 0,Y 170.238,Z 945.439,A -85,B 0,C 180,E1 8568.137,E2 8568.137} C_VEL
LIN {X 0,Y 169.969,Z 949.01,A -85,B 0,C 180,E1 8561.194,E2 8561.194} C_VEL
LIN {X 0,Y 170.741,Z 950.877,A -85,B 0,C 180,E1 8555.039,E2 8555.039} C_VEL
LIN {X 0,Y 171.274,Z 951.411,A -85,B 0,C 180,E1 8550.669,E2 8550.669} C_VEL
LIN {X 0,Y 171.013,Z 951.145,A -85,B 0,C 180,E1 8546.312,E2 8546.312} C_VEL
LIN {X 0,Y 170.316,Z 949.666,A -85,B 0,C 180,E1 8540.505,E2 8540.505} C_VEL
LIN {X 0,Y 170.453,Z 946.959,A -85,B 0,C 180,E1 8533.996,E2 8533.996} C_VEL
LIN {X 0,Y 173.084,Z 945.951,A -85,B 0,C 180,E1 8523.957,E2 8523.957} C_VEL
LIN {X 0,Y 180.438,Z 943.331,A -85,B 0,C 180,E1 8514.419,E2 8514.419} C_VEL
LIN {X 0,Y 196.51,Z 938.088,A -85,B 0,C 180,E1 8503.736,E2 8503.736} C_VEL
LIN {X 0,Y 214.673,Z 932.431,A -85,B 0,C 180,E1 8496.441,E2 8496.441} C_VEL
LIN {X 0,Y 200.309,Z 930.401,A -85,B 0,C 180,E1 8490.941,E2 8490.941} C_VEL
LIN {X 0,Y 189.197,Z 926.855,A -85,B 0,C 180,E1 8485.011,E2 8485.011} C_VEL
LIN {X 0,Y 180.649,Z 921.423,A -85,B 0,C 180,E1 8478.391,E2 8478.391} C_VEL
LIN {X 0,Y 175.206,Z 914.675,A -85,B 0,C 180,E1 8471.856,E2 8471.856} C_VEL
LIN {X 0,Y 171.943,Z 906.056,A -85,B 0,C 180,E1 8465.004,E2 8465.004} C_VEL
LIN {X 0,Y 170.634,Z 896.398,A -85,B 0,C 180,E1 8458.657,E2 8458.657} C_VEL
LIN {X 0,Y 170.574,Z 886.025,A -85,B 0,C 180,E1 8452.929,E2 8452.929} C_VEL
LIN {X 0,Y 171.537,Z 873.666,A -85,B 0,C 180,E1 8447.203,E2 8447.203} C_VEL
LIN {X 0,Y 172.27,Z 867.893,A -85,B 0,C 180,E1 8444.801,E2 8444.801} C_VEL
LIN {X 0,Y 173.563,Z 867.342,A -85,B 0,C 180,E1 8442.914,E2 8442.914} C_VEL
LIN {X 0,Y 175.531,Z 866.293,A -85,B 0,C 180,E1 8441.398,E2 8441.398} C_VEL
LIN {X 0,Y 177.882,Z 865.321,A -85,B 0,C 180,E1 8439.26,E2 8439.26} C_VEL
LIN {X 0,Y 179.964,Z 864.415,A -85,B 0,C 180,E1 8437.802,E2 8437.802} C_VEL
LIN {X 0,Y 188.449,Z 861.09,A -85,B 0,C 180,E1 8432.851,E2 8432.851} C_VEL
LIN {X 0,Y 195.136,Z 858.622,A -85,B 0,C 180,E1 8429.857,E2 8429.857} C_VEL
LIN {X 0,Y 201.808,Z 856.237,A -85,B 0,C 180,E1 8427.312,E2 8427.312} C_VEL
LIN {X 0,Y 210.529,Z 853.073,A -85,B 0,C 180,E1 8424.589,E2 8424.589} C_VEL
LIN {X 0,Y 219.938,Z 849.575,A -85,B 0,C 180,E1 8422.139,E2 8422.139} C_VEL
LIN {X 0,Y 227.467,Z 846.873,A -85,B 0,C 180,E1 8420.377,E2 8420.377} C_VEL
LIN {X 0,Y 216.58,Z 860.42,A -85,B 0,C 180,E1 8416.455,E2 8416.455} C_VEL
LIN {X 0,Y 206.231,Z 872.237,A -85,B 0,C 180,E1 8411.996,E2 8411.996} C_VEL
LIN {X 0,Y 196.607,Z 882.512,A -85,B 0,C 180,E1 8406.878,E2 8406.878} C_VEL
LIN {X 0,Y 188.064,Z 891.201,A -85,B 0,C 180,E1 8401.046,E2 8401.046} C_VEL
LIN {X 0,Y 180.987,Z 898.208,A -85,B 0,C 180,E1 8394.479,E2 8394.479} C_VEL
LIN {X 0,Y 176.12,Z 903.1,A -85,B 0,C 180,E1 8387.853,E2 8387.853} C_VEL
LIN {X 0,Y 172.956,Z 906.436,A -85,B 0,C 180,E1 8380.661,E2 8380.661} C_VEL
LIN {X 0,Y 171.582,Z 908.023,A -85,B 0,C 180,E1 8373.676,E2 8373.676} C_VEL
LIN {X 0,Y 171.513,Z 908.078,A -85,B 0,C 180,E1 8366.993,E2 8366.993} C_VEL
LIN {X 0,Y 172.643,Z 906.767,A -85,B 0,C 180,E1 8360.331,E2 8360.331} C_VEL
LIN {X 0,Y 175.352,Z 903.885,A -85,B 0,C 180,E1 8353.435,E2 8353.435} C_VEL
LIN {X 0,Y 179.86,Z 899.366,A -85,B 0,C 180,E1 8346.752,E2 8346.752} C_VEL
LIN {X 0,Y 186.196,Z 893.1,A -85,B 0,C 180,E1 8340.393,E2 8340.393} C_VEL
LIN {X 0,Y 194.323,Z 884.947,A -85,B 0,C 180,E1 8334.448,E2 8334.448} C_VEL
LIN {X 0,Y 203.592,Z 875.25,A -85,B 0,C 180,E1 8329.217,E2 8329.217} C_VEL
LIN {X 0,Y 213.642,Z 864.047,A -85,B 0,C 180,E1 8324.652,E2 8324.652} C_VEL
LIN {X 0,Y 224.14,Z 851.365,A -85,B 0,C 180,E1 8320.679,E2 8320.679} C_VEL
LIN {X 0,Y 234.176,Z 838.083,A -85,B 0,C 180,E1 8317.422,E2 8317.422} C_VEL
LIN {X 0,Y 244.444,Z 823.012,A -85,B 0,C 180,E1 8314.49,E2 8314.49} C_VEL
LIN {X 0,Y 254.128,Z 807.056,A -85,B 0,C 180,E1 8312.016,E2 8312.016} C_VEL
LIN {X 0,Y 263.412,Z 789.596,A -85,B 0,C 180,E1 8309.846,E2 8309.846} C_VEL
LIN {X 0,Y 271.811,Z 771.185,A -85,B 0,C 180,E1 8308.01,E2 8308.01} C_VEL
LIN {X 0,Y 278.845,Z 752.848,A -85,B 0,C 180,E1 8306.535,E2 8306.535} C_VEL
LIN {X 0,Y 285.181,Z 732.612,A -85,B 0,C 180,E1 8305.232,E2 8305.232} C_VEL
LIN {X 0,Y 291.329,Z 707.3,A -85,B 0,C 180,E1 8303.962,E2 8303.962} C_VEL
LIN {X 0,Y 299.972,Z 668.118,A -85,B 0,C 180,E1 8302.412,E2 8302.412} C_VEL
LIN {X 0,Y 308.109,Z 627.632,A -85,B 0,C 180,E1 8301.235,E2 8301.235} C_VEL
LIN {X 0,Y 315.744,Z 582.648,A -85,B 0,C 180,E1 8300.223,E2 8300.223} C_VEL
LIN {X 0,Y 321.542,Z 538.915,A -85,B 0,C 180,E1 8299.395,E2 8299.395} C_VEL
LIN {X 0,Y 328.061,Z 477.459,A -85,B 0,C 180,E1 8298.372,E2 8298.372} C_VEL
LIN {X 0,Y 330.414,Z 467.626,A -85,B 0,C 180,E1 8298.121,E2 8298.121} C_VEL
LIN {X 0,Y 328.768,Z 458.367,A -85,B 0,C 180,E1 8294.982,E2 8294.982} C_VEL
LIN {X 0,Y 327.363,Z 450.758,A -85,B 0,C 180,E1 8291.719,E2 8291.719} C_VEL
LIN {X 0,Y 326.436,Z 444.962,A -85,B 0,C 180,E1 8288.455,E2 8288.455} C_VEL
LIN {X 0,Y 326.01,Z 441.627,A -85,B 0,C 180,E1 8285.809,E2 8285.809} C_VEL
LIN {X 0,Y 326.136,Z 438.493,A -85,B 0,C 180,E1 8282.284,E2 8282.284} C_VEL
LIN {X 0,Y 327.092,Z 437.825,A -85,B 0,C 180,E1 8277.722,E2 8277.722} C_VEL
LIN {X 0,Y 327.678,Z 438.351,A -85,B 0,C 180,E1 8276.151,E2 8276.151} C_VEL
LIN {X 0,Y 327.603,Z 442.751,A -85,B 0,C 180,E1 8274.666,E2 8274.666} C_VEL
LIN {X 0,Y 327.409,Z 447.272,A -85,B 0,C 180,E1 8273.563,E2 8273.563} C_VEL
LIN {X 0,Y 326.255,Z 463.463,A -85,B 0,C 180,E1 8270.849,E2 8270.849} C_VEL
LIN {X 0,Y 326.362,Z 466.874,A -85,B 0,C 180,E1 8270.071,E2 8270.071} C_VEL
LIN {X 0,Y 326.397,Z 467.982,A -85,B 0,C 180,E1 8269.834,E2 8269.834} C_VEL
LIN {X 0,Y 312.259,Z 540.346,A -85,B 0,C 180,E1 8268.13,E2 8268.13} C_VEL
LIN {X 0,Y 305.28,Z 606.43,A -85,B 0,C 180,E1 8266.802,E2 8266.802} C_VEL
LIN {X 0,Y 299.526,Z 644.526,A -85,B 0,C 180,E1 8265.996,E2 8265.996} C_VEL
LIN {X 0,Y 292.237,Z 681.798,A -85,B 0,C 180,E1 8265.014,E2 8265.014} C_VEL
LIN {X 0,Y 284.118,Z 715.882,A -85,B 0,C 180,E1 8263.897,E2 8263.897} C_VEL
LIN {X 0,Y 274.729,Z 750.047,A -85,B 0,C 180,E1 8262.47,E2 8262.47} C_VEL
LIN {X 0,Y 265.655,Z 779.505,A -85,B 0,C 180,E1 8260.862,E2 8260.862} C_VEL
LIN {X 0,Y 258.296,Z 798.949,A -85,B 0,C 180,E1 8259.522,E2 8259.522} C_VEL
LIN {X 0,Y 249.49,Z 818.505,A -85,B 0,C 180,E1 8257.787,E2 8257.787} C_VEL
LIN {X 0,Y 240.123,Z 836.275,A -85,B 0,C 180,E1 8255.774,E2 8255.774} C_VEL
LIN {X 0,Y 229.924,Z 853.23,A -85,B 0,C 180,E1 8253.338,E2 8253.338} C_VEL
LIN {X 0,Y 219.29,Z 869.139,A -85,B 0,C 180,E1 8250.4,E2 8250.4} C_VEL
LIN {X 0,Y 208.732,Z 883.621,A -85,B 0,C 180,E1 8246.961,E2 8246.961} C_VEL
LIN {X 0,Y 198.182,Z 897.046,A -85,B 0,C 180,E1 8242.86,E2 8242.86} C_VEL
LIN {X 0,Y 187.748,Z 909.77,A -85,B 0,C 180,E1 8237.754,E2 8237.754} C_VEL
LIN {X 0,Y 178.855,Z 920.4,A -85,B 0,C 180,E1 8232.133,E2 8232.133} C_VEL
LIN {X 0,Y 171.118,Z 930.067,A -85,B 0,C 180,E1 8225.344,E2 8225.344} C_VEL
LIN {X 0,Y 165.718,Z 937.68,A -85,B 0,C 180,E1 8218.075,E2 8218.075} C_VEL
LIN {X 0,Y 162.719,Z 943.473,A -85,B 0,C 180,E1 8210.503,E2 8210.503} C_VEL
LIN {X 0,Y 161.934,Z 947.595,A -85,B 0,C 180,E1 8202.682,E2 8202.682} C_VEL
LIN {X 0,Y 162.628,Z 949.723,A -85,B 0,C 180,E1 8195.999,E2 8195.999} C_VEL
LIN {X 0,Y 163.282,Z 950.365,A -85,B 0,C 180,E1 8191.403,E2 8191.403} C_VEL
LIN {X 0,Y 163.17,Z 950.261,A -85,B 0,C 180,E1 8187.19,E2 8187.19} C_VEL
LIN {X 0,Y 162.418,Z 948.979,A -85,B 0,C 180,E1 8181.146,E2 8181.146} C_VEL
LIN {X 0,Y 162.552,Z 945.843,A -85,B 0,C 180,E1 8173.563,E2 8173.563} C_VEL
LIN {X 0,Y 162.923,Z 944.984,A -85,B 0,C 180,E1 8171.389,E2 8171.389} C_VEL
LIN {X 0,Y 167.484,Z 943.728,A -85,B 0,C 180,E1 8159.901,E2 8159.901} C_VEL
LIN {X 0,Y 177.688,Z 940.769,A -85,B 0,C 180,E1 8149.674,E2 8149.674} C_VEL
LIN {X 0,Y 197.239,Z 935.36,A -85,B 0,C 180,E1 8139.138,E2 8139.138} C_VEL
LIN {X 0,Y 204.404,Z 933.345,A -85,B 0,C 180,E1 8136.406,E2 8136.406} C_VEL
LIN {X 0,Y 190.818,Z 930.638,A -85,B 0,C 180,E1 8130.899,E2 8130.899} C_VEL
LIN {X 0,Y 179.821,Z 926.238,A -85,B 0,C 180,E1 8124.648,E2 8124.648} C_VEL
LIN {X 0,Y 171.811,Z 920.292,A -85,B 0,C 180,E1 8117.966,E2 8117.966} C_VEL
LIN {X 0,Y 166.376,Z 912.489,A -85,B 0,C 180,E1 8110.737,E2 8110.737} C_VEL
LIN {X 0,Y 163.582,Z 903.556,A -85,B 0,C 180,E1 8103.855,E2 8103.855} C_VEL
LIN {X 0,Y 162.558,Z 893.783,A -85,B 0,C 180,E1 8097.532,E2 8097.532} C_VEL
LIN {X 0,Y 162.772,Z 881.994,A -85,B 0,C 180,E1 8091.166,E2 8091.166} C_VEL
LIN {X 0,Y 163.456,Z 874.182,A -85,B 0,C 180,E1 8087.458,E2 8087.458} C_VEL
LIN {X 0,Y 164.692,Z 873.5,A -85,B 0,C 180,E1 8085.227,E2 8085.227} C_VEL
LIN {X 0,Y 166.338,Z 872.586,A -85,B 0,C 180,E1 8083.589,E2 8083.589} C_VEL
LIN {X 0,Y 168.481,Z 871.593,A -85,B 0,C 180,E1 8081.308,E2 8081.308} C_VEL
LIN {X 0,Y 169.996,Z 870.896,A -85,B 0,C 180,E1 8080.053,E2 8080.053} C_VEL
LIN {X 0,Y 173.185,Z 869.561,A -85,B 0,C 180,E1 8077.601,E2 8077.601} C_VEL
LIN {X 0,Y 178.171,Z 867.644,A -85,B 0,C 180,E1 8074.397,E2 8074.397} C_VEL
LIN {X 0,Y 183.824,Z 865.611,A -85,B 0,C 180,E1 8071.401,E2 8071.401} C_VEL
LIN {X 0,Y 196.302,Z 861.336,A -85,B 0,C 180,E1 8066.275,E2 8066.275} C_VEL
LIN {X 0,Y 213.962,Z 855.173,A -85,B 0,C 180,E1 8061.229,E2 8061.229} C_VEL
LIN {X 0,Y 217.717,Z 853.818,A -85,B 0,C 180,E1 8060.381,E2 8060.381} C_VEL
LIN {X 0,Y 206.463,Z 866.757,A -85,B 0,C 180,E1 8056.168,E2 8056.168} C_VEL
LIN {X 0,Y 195.999,Z 877.812,A -85,B 0,C 180,E1 8051.416,E2 8051.416} C_VEL
LIN {X 0,Y 186.64,Z 887.075,A -85,B 0,C 180,E1 8046.108,E2 8046.108} C_VEL
LIN {X 0,Y 178.646,Z 894.647,A -85,B 0,C 180,E1 8040.248,E2 8040.248} C_VEL
LIN {X 0,Y 172.072,Z 900.773,A -85,B 0,C 180,E1 8033.638,E2 8033.638} C_VEL
LIN {X 0,Y 167.41,Z 905.164,A -85,B 0,C 180,E1 8026.66,E2 8026.66} C_VEL
LIN {X 0,Y 164.64,Z 907.919,A -85,B 0,C 180,E1 8019.438,E2 8019.438} C_VEL
LIN {X 0,Y 163.516,Z 909.125,A -85,B 0,C 180,E1 8012.103,E2 8012.103} C_VEL
LIN {X 0,Y 163.758,Z 908.882,A -85,B 0,C 180,E1 8005.096,E2 8005.096} C_VEL
LIN {X 0,Y 165.345,Z 907.279,A -85,B 0,C 180,E1 7998.135,E2 7998.135} C_VEL
LIN {X 0,Y 168.914,Z 903.828,A -85,B 0,C 180,E1 7990.641,E2 7990.641} C_VEL
LIN {X 0,Y 174.289,Z 898.843,A -85,B 0,C 180,E1 7983.785,E2 7983.785} C_VEL
LIN {X 0,Y 181.575,Z 892.061,A -85,B 0,C 180,E1 7977.34,E2 7977.34} C_VEL
LIN {X 0,Y 190.656,Z 883.332,A -85,B 0,C 180,E1 7971.385,E2 7971.385} C_VEL
LIN {X 0,Y 200.81,Z 873.018,A -85,B 0,C 180,E1 7966.202,E2 7966.202} C_VEL
LIN {X 0,Y 211.3,Z 861.561,A -85,B 0,C 180,E1 7961.854,E2 7961.854} C_VEL
LIN {X 0,Y 222.217,Z 848.54,A -85,B 0,C 180,E1 7958.054,E2 7958.054} C_VEL
LIN {X 0,Y 232.801,Z 834.608,A -85,B 0,C 180,E1 7954.88,E2 7954.88} C_VEL
LIN {X 0,Y 243.208,Z 819.289,A -85,B 0,C 180,E1 7952.122,E2 7952.122} C_VEL
LIN {X 0,Y 252.927,Z 803.13,A -85,B 0,C 180,E1 7949.803,E2 7949.803} C_VEL
LIN {X 0,Y 261.796,Z 786.253,A -85,B 0,C 180,E1 7947.849,E2 7947.849} C_VEL
LIN {X 0,Y 270.198,Z 767.496,A -85,B 0,C 180,E1 7946.102,E2 7946.102} C_VEL
LIN {X 0,Y 277.309,Z 748.444,A -85,B 0,C 180,E1 7944.683,E2 7944.683} C_VEL
LIN {X 0,Y 283.179,Z 728.923,A -85,B 0,C 180,E1 7943.516,E2 7943.516} C_VEL
LIN {X 0,Y 292.148,Z 691.357,A -85,B 0,C 180,E1 7941.802,E2 7941.802} C_VEL
LIN {X 0,Y 300.79,Z 651.633,A -85,B 0,C 180,E1 7940.445,E2 7940.445} C_VEL
LIN {X 0,Y 309.071,Z 608.575,A -85,B 0,C 180,E1 7939.379,E2 7939.379} C_VEL
LIN {X 0,Y 315.944,Z 564.301,A -85,B 0,C 180,E1 7938.479,E2 7938.479} C_VEL
LIN {X 0,Y 321.34,Z 518.138,A -85,B 0,C 180,E1 7937.685,E2 7937.685} C_VEL
LIN {X 0,Y 325.459,Z 480.137,A -85,B 0,C 180,E1 7937.07,E2 7937.07} C_VEL
LIN {X 0,Y 327.356,Z 472.231,A -85,B 0,C 180,E1 7936.868,E2 7936.868} C_VEL
LIN {X 0,Y 326.031,Z 463.911,A -85,B 0,C 180,E1 7933.886,E2 7933.886} C_VEL
LIN {X 0,Y 324.966,Z 457.487,A -85,B 0,C 180,E1 7930.998,E2 7930.998} C_VEL
LIN {X 0,Y 324.283,Z 452.166,A -85,B 0,C 180,E1 7927.887,E2 7927.887} C_VEL
LIN {X 0,Y 324.015,Z 449.197,A -85,B 0,C 180,E1 7925.49,E2 7925.49} C_VEL
LIN {X 0,Y 324.198,Z 446.224,A -85,B 0,C 180,E1 7922.121,E2 7922.121} C_VEL
LIN {X 0,Y 325.29,Z 445.62,A -85,B 0,C 180,E1 7917.71,E2 7917.71} C_VEL
LIN {X 0,Y 325.711,Z 446.095,A -85,B 0,C 180,E1 7916.48,E2 7916.48} C_VEL
LIN {X 0,Y 325.714,Z 457.481,A -85,B 0,C 180,E1 7912.769,E2 7912.769} C_VEL
LIN {X 0,Y 326.362,Z 466.874,A -85,B 0,C 180,E1 7910.071,E2 7910.071} C_VEL
LIN {X 0,Y 326.236,Z 469.482,A -85,B 0,C 180,E1 7909.694,E2 7909.694} C_VEL
LIN {X 0,Y 325.497,Z 473.821,A -85,B 0,C 180,E1 7909.518,E2 7909.518} C_VEL
LIN {X 0,Y 323.928,Z 480.199,A -85,B 0,C 180,E1 7909.645,E2 7909.645} C_VEL
LIN {X 0,Y 319.801,Z 494.115,A -85,B 0,C 180,E1 7910.402,E2 7910.402} C_VEL
LIN {X 0,Y 318.284,Z 500.243,A -85,B 0,C 180,E1 7910.5,E2 7910.5} C_VEL
LIN {X 0,Y 318.03,Z 501.48,A -85,B 0,C 180,E1 7910.48,E2 7910.48} C_VEL
LIN {X 0,Y 310.898,Z 537.494,A -85,B 0,C 180,E1 7909.633,E2 7909.633} C_VEL
LIN {X 0,Y 303.693,Z 603.933,A -85,B 0,C 180,E1 7908.32,E2 7908.32} C_VEL
LIN {X 0,Y 297.888,Z 641.792,A -85,B 0,C 180,E1 7907.542,E2 7907.542} C_VEL
LIN {X 0,Y 290.39,Z 679.604,A -85,B 0,C 180,E1 7906.587,E2 7906.587} C_VEL
LIN {X 0,Y 281.841,Z 714.965,A -85,B 0,C 180,E1 7905.475,E2 7905.475} C_VEL
LIN {X 0,Y 272.159,Z 749.508,A -85,B 0,C 180,E1 7904.08,E2 7904.08} C_VEL
LIN {X 0,Y 262.796,Z 779.154,A -85,B 0,C 180,E1 7902.507,E2 7902.507} C_VEL
LIN {X 0,Y 255.108,Z 798.754,A -85,B 0,C 180,E1 7901.183,E2 7901.183} C_VEL
LIN {X 0,Y 246.068,Z 818.016,A -85,B 0,C 180,E1 7899.493,E2 7899.493} C_VEL
LIN {X 0,Y 236.339,Z 835.816,A -85,B 0,C 180,E1 7897.512,E2 7897.512} C_VEL
LIN {X 0,Y 225.529,Z 853.14,A -85,B 0,C 180,E1 7895.048,E2 7895.048} C_VEL
LIN {X 0,Y 213.681,Z 870.088,A -85,B 0,C 180,E1 7891.892,E2 7891.892} C_VEL
LIN {X 0,Y 202.24,Z 884.969,A -85,B 0,C 180,E1 7888.253,E2 7888.253} C_VEL
LIN {X 0,Y 190.763,Z 898.788,A -85,B 0,C 180,E1 7883.823,E2 7883.823} C_VEL
LIN {X 0,Y 180.044,Z 911.037,A -85,B 0,C 180,E1 7878.567,E2 7878.567} C_VEL
LIN {X 0,Y 170.49,Z 921.75,A -85,B 0,C 180,E1 7872.411,E2 7872.411} C_VEL
LIN {X 0,Y 162.49,Z 931.148,A -85,B 0,C 180,E1 7865.072,E2 7865.072} C_VEL
LIN {X 0,Y 157.152,Z 938.44,A -85,B 0,C 180,E1 7857.265,E2 7857.265} C_VEL
LIN {X 0,Y 154.396,Z 943.938,A -85,B 0,C 180,E1 7849,E2 7849} C_VEL
LIN {X 0,Y 154.042,Z 947.377,A -85,B 0,C 180,E1 7841.229,E2 7841.229} C_VEL
LIN {X 0,Y 154.925,Z 949.061,A -85,B 0,C 180,E1 7834.442,E2 7834.442} C_VEL
LIN {X 0,Y 155.419,Z 949.442,A -85,B 0,C 180,E1 7830,E2 7830} C_VEL
LIN {X 0,Y 154.951,Z 948.992,A -85,B 0,C 180,E1 7825.188,E2 7825.188} C_VEL
LIN {X 0,Y 154.303,Z 947.253,A -85,B 0,C 180,E1 7818.411,E2 7818.411} C_VEL
LIN {X 0,Y 155.177,Z 943.6,A -85,B 0,C 180,E1 7810.423,E2 7810.423} C_VEL
LIN {X 0,Y 155.685,Z 942.909,A -85,B 0,C 180,E1 7808.633,E2 7808.633} C_VEL
LIN {X 0,Y 162.106,Z 941.586,A -85,B 0,C 180,E1 7796.28,E2 7796.28} C_VEL
LIN {X 0,Y 175.717,Z 938.278,A -85,B 0,C 180,E1 7785.121,E2 7785.121} C_VEL
LIN {X 0,Y 194.155,Z 933.809,A -85,B 0,C 180,E1 7776.379,E2 7776.379} C_VEL
LIN {X 0,Y 180.797,Z 930.272,A -85,B 0,C 180,E1 7770.584,E2 7770.584} C_VEL
LIN {X 0,Y 170.046,Z 924.983,A -85,B 0,C 180,E1 7763.937,E2 7763.937} C_VEL
LIN {X 0,Y 162.406,Z 918.195,A -85,B 0,C 180,E1 7756.82,E2 7756.82} C_VEL
LIN {X 0,Y 157.612,Z 909.934,A -85,B 0,C 180,E1 7749.494,E2 7749.494} C_VEL
LIN {X 0,Y 155.194,Z 900.202,A -85,B 0,C 180,E1 7742.215,E2 7742.215} C_VEL
LIN {X 0,Y 154.524,Z 889.524,A -85,B 0,C 180,E1 7735.546,E2 7735.546} C_VEL
LIN {X 0,Y 154.874,Z 880.228,A -85,B 0,C 180,E1 7730.524,E2 7730.524} C_VEL
LIN {X 0,Y 155.771,Z 879.544,A -85,B 0,C 180,E1 7728.147,E2 7728.147} C_VEL
LIN {X 0,Y 157.17,Z 878.655,A -85,B 0,C 180,E1 7726.385,E2 7726.385} C_VEL
LIN {X 0,Y 159.294,Z 877.528,A -85,B 0,C 180,E1 7723.592,E2 7723.592} C_VEL
LIN {X 0,Y 163.019,Z 875.829,A -85,B 0,C 180,E1 7719.911,E2 7719.911} C_VEL
LIN {X 0,Y 167.509,Z 874.038,A -85,B 0,C 180,E1 7716.426,E2 7716.426} C_VEL
LIN {X 0,Y 177.965,Z 870.352,A -85,B 0,C 180,E1 7710.368,E2 7710.368} C_VEL
LIN {X 0,Y 192.867,Z 865.444,A -85,B 0,C 180,E1 7704.504,E2 7704.504} C_VEL
LIN {X 0,Y 207.636,Z 860.681,A -85,B 0,C 180,E1 7700.291,E2 7700.291} C_VEL
LIN {X 0,Y 196.368,Z 872.639,A -85,B 0,C 180,E1 7695.887,E2 7695.887} C_VEL
LIN {X 0,Y 185.576,Z 883.186,A -85,B 0,C 180,E1 7690.689,E2 7690.689} C_VEL
LIN {X 0,Y 175.811,Z 892.134,A -85,B 0,C 180,E1 7684.662,E2 7684.662} C_VEL
LIN {X 0,Y 167.874,Z 899.118,A -85,B 0,C 180,E1 7678.07,E2 7678.07} C_VEL
LIN {X 0,Y 161.913,Z 904.303,A -85,B 0,C 180,E1 7670.989,E2 7670.989} C_VEL
LIN {X 0,Y 157.98,Z 907.815,A -85,B 0,C 180,E1 7663.544,E2 7663.544} C_VEL
LIN {X 0,Y 155.961,Z 909.742,A -85,B 0,C 180,E1 7655.888,E2 7655.888} C_VEL
LIN {X 0,Y 155.547,Z 910.174,A -85,B 0,C 180,E1 7648.527,E2 7648.527} C_VEL
LIN {X 0,Y 156.513,Z 909.256,A -85,B 0,C 180,E1 7641.181,E2 7641.181} C_VEL
LIN {X 0,Y 159.212,Z 906.786,A -85,B 0,C 180,E1 7633.584,E2 7633.584} C_VEL
LIN {X 0,Y 164.178,Z 902.442,A -85,B 0,C 180,E1 7625.918,E2 7625.918} C_VEL
LIN {X 0,Y 170.972,Z 896.543,A -85,B 0,C 180,E1 7619.026,E2 7619.026} C_VEL
LIN {X 0,Y 179.703,Z 888.775,A -85,B 0,C 180,E1 7612.664,E2 7612.664} C_VEL
LIN {X 0,Y 189.691,Z 879.429,A -85,B 0,C 180,E1 7607.113,E2 7607.113} C_VEL
LIN {X 0,Y 200.352,Z 868.737,A -85,B 0,C 180,E1 7602.386,E2 7602.386} C_VEL
LIN {X 0,Y 211.504,Z 856.553,A -85,B 0,C 180,E1 7598.301,E2 7598.301} C_VEL
LIN {X 0,Y 222.123,Z 843.831,A -85,B 0,C 180,E1 7594.988,E2 7594.988} C_VEL
LIN {X 0,Y 233.302,Z 828.879,A -85,B 0,C 180,E1 7591.941,E2 7591.941} C_VEL
LIN {X 0,Y 243.856,Z 812.959,A -85,B 0,C 180,E1 7589.388,E2 7589.388} C_VEL
LIN {X 0,Y 253.878,Z 795.636,A -85,B 0,C 180,E1 7587.185,E2 7587.185} C_VEL
LIN {X 0,Y 262.798,Z 777.688,A -85,B 0,C 180,E1 7585.36,E2 7585.36} C_VEL
LIN {X 0,Y 270.565,Z 759.168,A -85,B 0,C 180,E1 7583.844,E2 7583.844} C_VEL
LIN {X 0,Y 277.219,Z 739.86,A -85,B 0,C 180,E1 7582.578,E2 7582.578} C_VEL
LIN {X 0,Y 282.976,Z 718.593,A -85,B 0,C 180,E1 7581.467,E2 7581.467} C_VEL
LIN {X 0,Y 291.879,Z 681.09,A -85,B 0,C 180,E1 7579.925,E2 7579.925} C_VEL
LIN {X 0,Y 300.204,Z 642.664,A -85,B 0,C 180,E1 7578.745,E2 7578.745} C_VEL
LIN {X 0,Y 308.37,Z 599.066,A -85,B 0,C 180,E1 7577.752,E2 7577.752} C_VEL
LIN {X 0,Y 314.798,Z 555.878,A -85,B 0,C 180,E1 7576.931,E2 7576.931} C_VEL
LIN {X 0,Y 322.131,Z 488.972,A -85,B 0,C 180,E1 7575.854,E2 7575.854} C_VEL
LIN {X 0,Y 323.313,Z 481.69,A -85,B 0,C 180,E1 7575.723,E2 7575.723} C_VEL
LIN {X 0,Y 324.454,Z 476.957,A -85,B 0,C 180,E1 7575.598,E2 7575.598} C_VEL
LIN {X 0,Y 323.375,Z 469.3,A -85,B 0,C 180,E1 7572.682,E2 7572.682} C_VEL
LIN {X 0,Y 322.503,Z 462.664,A -85,B 0,C 180,E1 7569.458,E2 7569.458} C_VEL
LIN {X 0,Y 322.062,Z 458.355,A -85,B 0,C 180,E1 7566.543,E2 7566.543} C_VEL
LIN {X 0,Y 322.023,Z 456.468,A -85,B 0,C 180,E1 7564.809,E2 7564.809} C_VEL
LIN {X 0,Y 322.392,Z 453.985,A -85,B 0,C 180,E1 7561.955,E2 7561.955} C_VEL
LIN {X 0,Y 323.478,Z 453.423,A -85,B 0,C 180,E1 7557.52,E2 7557.52} C_VEL
LIN {X 0,Y 323.726,Z 453.75,A -85,B 0,C 180,E1 7556.857,E2 7556.857} C_VEL
LIN {X 0,Y 323.619,Z 464.22,A -85,B 0,C 180,E1 7553.436,E2 7553.436} C_VEL
LIN {X 0,Y 323.99,Z 472.347,A -85,B 0,C 180,E1 7551.126,E2 7551.126} C_VEL
LIN {X 0,Y 318.03,Z 501.48,A -85,B 0,C 180,E1 7550.48,E2 7550.48} C_VEL
LIN {X 0,Y 316.548,Z 507.968,A -85,B 0,C 180,E1 7550.482,E2 7550.482} C_VEL
LIN {X 0,Y 311.017,Z 528.159,A -85,B 0,C 180,E1 7551.159,E2 7551.159} C_VEL
LIN {X 0,Y 309.629,Z 535.804,A -85,B 0,C 180,E1 7551.126,E2 7551.126} C_VEL
LIN {X 0,Y 302.321,Z 601.428,A -85,B 0,C 180,E1 7549.853,E2 7549.853} C_VEL
LIN {X 0,Y 296.532,Z 638.71,A -85,B 0,C 180,E1 7549.111,E2 7549.111} C_VEL
LIN {X 0,Y 289.033,Z 676.098,A -85,B 0,C 180,E1 7548.212,E2 7548.212} C_VEL
LIN {X 0,Y 280.532,Z 711.081,A -85,B 0,C 180,E1 7547.174,E2 7547.174} C_VEL
LIN {X 0,Y 270.691,Z 746.056,A -85,B 0,C 180,E1 7545.844,E2 7545.844} C_VEL
LIN {X 0,Y 261.149,Z 775.901,A -85,B 0,C 180,E1 7544.354,E2 7544.354} C_VEL
LIN {X 0,Y 253.42,Z 795.529,A -85,B 0,C 180,E1 7543.098,E2 7543.098} C_VEL
LIN {X 0,Y 244.549,Z 814.389,A -85,B 0,C 180,E1 7541.546,E2 7541.546} C_VEL
LIN {X 0,Y 234.584,Z 832.421,A -85,B 0,C 180,E1 7539.673,E2 7539.673} C_VEL
LIN {X 0,Y 223.313,Z 850.179,A -85,B 0,C 180,E1 7537.275,E2 7537.275} C_VEL
LIN {X 0,Y 211.744,Z 866.408,A -85,B 0,C 180,E1 7534.413,E2 7534.413} C_VEL
LIN {X 0,Y 199.981,Z 881.31,A -85,B 0,C 180,E1 7530.988,E2 7530.988} C_VEL
LIN {X 0,Y 187.826,Z 895.418,A -85,B 0,C 180,E1 7526.698,E2 7526.698} C_VEL
LIN {X 0,Y 176.834,Z 907.448,A -85,B 0,C 180,E1 7521.809,E2 7521.809} C_VEL
LIN {X 0,Y 166.405,Z 918.484,A -85,B 0,C 180,E1 7515.812,E2 7515.812} C_VEL
LIN {X 0,Y 157.691,Z 927.835,A -85,B 0,C 180,E1 7508.883,E2 7508.883} C_VEL
LIN {X 0,Y 151.147,Z 935.497,A -85,B 0,C 180,E1 7501.064,E2 7501.064} C_VEL
LIN {X 0,Y 147.215,Z 941.475,A -85,B 0,C 180,E1 7492.524,E2 7492.524} C_VEL
LIN {X 0,Y 145.987,Z 945.594,A -85,B 0,C 180,E1 7483.87,E2 7483.87} C_VEL
LIN {X 0,Y 146.665,Z 947.759,A -85,B 0,C 180,E1 7476.262,E2 7476.262} C_VEL
LIN {X 0,Y 147.416,Z 948.383,A -85,B 0,C 180,E1 7471.166,E2 7471.166} C_VEL
LIN {X 0,Y 147.236,Z 948.249,A -85,B 0,C 180,E1 7466.885,E2 7466.885} C_VEL
LIN {X 0,Y 146.413,Z 946.928,A -85,B 0,C 180,E1 7460.169,E2 7460.169} C_VEL
LIN {X 0,Y 146.896,Z 943.753,A -85,B 0,C 180,E1 7451.753,E2 7451.753} C_VEL
LIN {X 0,Y 148.736,Z 940.738,A -85,B 0,C 180,E1 7445.79,E2 7445.79} C_VEL
LIN {X 0,Y 155.377,Z 939.69,A -85,B 0,C 180,E1 7434.607,E2 7434.607} C_VEL
LIN {X 0,Y 171.57,Z 936.487,A -85,B 0,C 180,E1 7422.256,E2 7422.256} C_VEL
LIN {X 0,Y 184.071,Z 933.865,A -85,B 0,C 180,E1 7416.412,E2 7416.412} C_VEL
LIN {X 0,Y 170.784,Z 929.414,A -85,B 0,C 180,E1 7410.232,E2 7410.232} C_VEL
LIN {X 0,Y 160.311,Z 923.283,A -85,B 0,C 180,E1 7403.138,E2 7403.138} C_VEL
LIN {X 0,Y 152.813,Z 915.245,A -85,B 0,C 180,E1 7395.173,E2 7395.173} C_VEL
LIN {X 0,Y 148.626,Z 905.995,A -85,B 0,C 180,E1 7387.344,E2 7387.344} C_VEL
LIN {X 0,Y 146.843,Z 895.8,A -85,B 0,C 180,E1 7380,E2 7380} C_VEL
LIN {X 0,Y 146.572,Z 886.134,A -85,B 0,C 180,E1 7373.93,E2 7373.93} C_VEL
LIN {X 0,Y 147.399,Z 885.194,A -85,B 0,C 180,E1 7371.024,E2 7371.024} C_VEL
LIN {X 0,Y 148.317,Z 884.486,A -85,B 0,C 180,E1 7369.512,E2 7369.512} C_VEL
LIN {X 0,Y 149.995,Z 883.391,A -85,B 0,C 180,E1 7366.508,E2 7366.508} C_VEL
LIN {X 0,Y 153.551,Z 881.562,A -85,B 0,C 180,E1 7362.178,E2 7362.178} C_VEL
LIN {X 0,Y 157.086,Z 880.085,A -85,B 0,C 180,E1 7358.726,E2 7358.726} C_VEL
LIN {X 0,Y 167.216,Z 876.434,A -85,B 0,C 180,E1 7351.81,E2 7351.81} C_VEL
LIN {X 0,Y 180.712,Z 872.139,A -85,B 0,C 180,E1 7345.641,E2 7345.641} C_VEL
LIN {X 0,Y 196.903,Z 867.132,A -85,B 0,C 180,E1 7340.522,E2 7340.522} C_VEL
LIN {X 0,Y 197.669,Z 866.971,A -85,B 0,C 180,E1 7340.254,E2 7340.254} C_VEL
LIN {X 0,Y 186.217,Z 878.185,A -85,B 0,C 180,E1 7335.573,E2 7335.573} C_VEL
LIN {X 0,Y 175.474,Z 887.891,A -85,B 0,C 180,E1 7330.084,E2 7330.084} C_VEL
LIN {X 0,Y 165.864,Z 896.049,A -85,B 0,C 180,E1 7323.684,E2 7323.684} C_VEL
LIN {X 0,Y 157.881,Z 902.574,A -85,B 0,C 180,E1 7316.316,E2 7316.316} C_VEL
LIN {X 0,Y 152.208,Z 907.194,A -85,B 0,C 180,E1 7308.381,E2 7308.381} C_VEL
LIN {X 0,Y 148.973,Z 909.931,A -85,B 0,C 180,E1 7300.441,E2 7300.441} C_VEL
LIN {X 0,Y 147.652,Z 911.127,A -85,B 0,C 180,E1 7292.329,E2 7292.329} C_VEL
LIN {X 0,Y 147.938,Z 910.887,A -85,B 0,C 180,E1 7284.571,E2 7284.571} C_VEL
LIN {X 0,Y 149.799,Z 909.291,A -85,B 0,C 180,E1 7276.883,E2 7276.883} C_VEL
LIN {X 0,Y 153.953,Z 905.858,A -85,B 0,C 180,E1 7268.672,E2 7268.672} C_VEL
LIN {X 0,Y 160.113,Z 900.891,A -85,B 0,C 180,E1 7261.259,E2 7261.259} C_VEL
LIN {X 0,Y 168.341,Z 894.131,A -85,B 0,C 180,E1 7254.403,E2 7254.403} C_VEL
LIN {X 0,Y 177.935,Z 885.906,A -85,B 0,C 180,E1 7248.464,E2 7248.464} C_VEL
LIN {X 0,Y 188.44,Z 876.302,A -85,B 0,C 180,E1 7243.369,E2 7243.369} C_VEL
LIN {X 0,Y 200.111,Z 864.677,A -85,B 0,C 180,E1 7238.787,E2 7238.787} C_VEL
LIN {X 0,Y 212.085,Z 851.535,A -85,B 0,C 180,E1 7234.882,E2 7234.882} C_VEL
LIN {X 0,Y 223.366,Z 837.762,A -85,B 0,C 180,E1 7231.731,E2 7231.731} C_VEL
LIN {X 0,Y 234.763,Z 822.076,A -85,B 0,C 180,E1 7228.932,E2 7228.932} C_VEL
LIN {X 0,Y 245.041,Z 806,A -85,B 0,C 180,E1 7226.667,E2 7226.667} C_VEL
LIN {X 0,Y 254.379,Z 789.217,A -85,B 0,C 180,E1 7224.771,E2 7224.771} C_VEL
LIN {X 0,Y 262.679,Z 771.838,A -85,B 0,C 180,E1 7223.18,E2 7223.18} C_VEL
LIN {X 0,Y 270.267,Z 752.827,A -85,B 0,C 180,E1 7221.781,E2 7221.781} C_VEL
LIN {X 0,Y 276.477,Z 733.625,A -85,B 0,C 180,E1 7220.646,E2 7220.646} C_VEL
LIN {X 0,Y 285.763,Z 697.265,A -85,B 0,C 180,E1 7219,E2 7219} C_VEL
LIN {X 0,Y 294.593,Z 658.964,A -85,B 0,C 180,E1 7217.701,E2 7217.701} C_VEL
LIN {X 0,Y 302.738,Z 618.995,A -85,B 0,C 180,E1 7216.721,E2 7216.721} C_VEL
LIN {X 0,Y 309.89,Z 576.441,A -85,B 0,C 180,E1 7215.877,E2 7215.877} C_VEL
LIN {X 0,Y 315.416,Z 533.436,A -85,B 0,C 180,E1 7215.152,E2 7215.152} C_VEL
LIN {X 0,Y 320.745,Z 485.656,A -85,B 0,C 180,E1 7214.409,E2 7214.409} C_VEL
LIN {X 0,Y 321.688,Z 481.786,A -85,B 0,C 180,E1 7214.307,E2 7214.307} C_VEL
LIN {X 0,Y 320.793,Z 474.307,A -85,B 0,C 180,E1 7211.234,E2 7211.234} C_VEL
LIN {X 0,Y 320.211,Z 468.481,A -85,B 0,C 180,E1 7208.078,E2 7208.078} C_VEL
LIN {X 0,Y 320.057,Z 464.479,A -85,B 0,C 180,E1 7205.018,E2 7205.018} C_VEL
LIN {X 0,Y 320.519,Z 461.73,A -85,B 0,C 180,E1 7201.788,E2 7201.788} C_VEL
LIN {X 0,Y 321.663,Z 461.217,A -85,B 0,C 180,E1 7197.506,E2 7197.506} C_VEL
LIN {X 0,Y 321.72,Z 461.658,A -85,B 0,C 180,E1 7197.15,E2 7197.15} C_VEL
LIN {X 0,Y 321.499,Z 471.093,A -85,B 0,C 180,E1 7194.064,E2 7194.064} C_VEL
LIN {X 0,Y 321.594,Z 476.923,A -85,B 0,C 180,E1 7192.43,E2 7192.43} C_VEL
LIN {X 0,Y 309.776,Z 534.416,A -85,B 0,C 180,E1 7191.154,E2 7191.154} C_VEL
LIN {X 0,Y 309.629,Z 535.804,A -85,B 0,C 180,E1 7191.126,E2 7191.126} C_VEL
LIN {X 0,Y 308.646,Z 543.505,A -85,B 0,C 180,E1 7191.156,E2 7191.156} C_VEL
LIN {X 0,Y 305.429,Z 564.115,A -85,B 0,C 180,E1 7191.923,E2 7191.923} C_VEL
LIN {X 0,Y 304.602,Z 570.726,A -85,B 0,C 180,E1 7191.937,E2 7191.937} C_VEL
LIN {X 0,Y 299.515,Z 610.459,A -85,B 0,C 180,E1 7191.172,E2 7191.172} C_VEL
LIN {X 0,Y 293.011,Z 648.006,A -85,B 0,C 180,E1 7190.43,E2 7190.43} C_VEL
LIN {X 0,Y 284.888,Z 685.595,A -85,B 0,C 180,E1 7189.509,E2 7189.509} C_VEL
LIN {X 0,Y 276.271,Z 719.212,A -85,B 0,C 180,E1 7188.495,E2 7188.495} C_VEL
LIN {X 0,Y 266.563,Z 752.045,A -85,B 0,C 180,E1 7187.231,E2 7187.231} C_VEL
LIN {X 0,Y 258.109,Z 777.266,A -85,B 0,C 180,E1 7185.963,E2 7185.963} C_VEL
LIN {X 0,Y 249.689,Z 797.475,A -85,B 0,C 180,E1 7184.675,E2 7184.675} C_VEL
LIN {X 0,Y 240.334,Z 816.295,A -85,B 0,C 180,E1 7183.116,E2 7183.116} C_VEL
LIN {X 0,Y 229.783,Z 834.418,A -85,B 0,C 180,E1 7181.216,E2 7181.216} C_VEL
LIN {X 0,Y 218.185,Z 851.818,A -85,B 0,C 180,E1 7178.842,E2 7178.842} C_VEL
LIN {X 0,Y 206.701,Z 867.164,A -85,B 0,C 180,E1 7176.101,E2 7176.101} C_VEL
LIN {X 0,Y 195.127,Z 881.149,A -85,B 0,C 180,E1 7172.867,E2 7172.867} C_VEL
LIN {X 0,Y 182.758,Z 894.872,A -85,B 0,C 180,E1 7168.684,E2 7168.684} C_VEL
LIN {X 0,Y 170.534,Z 907.555,A -85,B 0,C 180,E1 7163.443,E2 7163.443} C_VEL
LIN {X 0,Y 159.443,Z 918.511,A -85,B 0,C 180,E1 7157.199,E2 7157.199} C_VEL
LIN {X 0,Y 150.43,Z 927.504,A -85,B 0,C 180,E1 7150.147,E2 7150.147} C_VEL
LIN {X 0,Y 143.494,Z 935.031,A -85,B 0,C 180,E1 7141.977,E2 7141.977} C_VEL
LIN {X 0,Y 139.264,Z 940.973,A -85,B 0,C 180,E1 7132.812,E2 7132.812} C_VEL
LIN {X 0,Y 138.021,Z 944.864,A -85,B 0,C 180,E1 7123.831,E2 7123.831} C_VEL
LIN {X 0,Y 138.775,Z 946.888,A -85,B 0,C 180,E1 7115.789,E2 7115.789} C_VEL
LIN {X 0,Y 139.501,Z 947.405,A -85,B 0,C 180,E1 7110.821,E2 7110.821} C_VEL
LIN {X 0,Y 139.209,Z 947.209,A -85,B 0,C 180,E1 7106.293,E2 7106.293} C_VEL
LIN {X 0,Y 138.396,Z 945.673,A -85,B 0,C 180,E1 7098.751,E2 7098.751} C_VEL
LIN {X 0,Y 139.297,Z 942.315,A -85,B 0,C 180,E1 7089.845,E2 7089.845} C_VEL
LIN {X 0,Y 142.085,Z 938.515,A -85,B 0,C 180,E1 7082.779,E2 7082.779} C_VEL
LIN {X 0,Y 151.455,Z 937.285,A -85,B 0,C 180,E1 7070.179,E2 7070.179} C_VEL
LIN {X 0,Y 167.908,Z 934.507,A -85,B 0,C 180,E1 7059.272,E2 7059.272} C_VEL
LIN {X 0,Y 173.977,Z 933.459,A -85,B 0,C 180,E1 7056.441,E2 7056.441} C_VEL
LIN {X 0,Y 160.793,Z 928.115,A -85,B 0,C 180,E1 7049.833,E2 7049.833} C_VEL
LIN {X 0,Y 150.628,Z 921.136,A -85,B 0,C 180,E1 7042.233,E2 7042.233} C_VEL
LIN {X 0,Y 143.831,Z 912.629,A -85,B 0,C 180,E1 7034.082,E2 7034.082} C_VEL
LIN {X 0,Y 140.181,Z 903.096,A -85,B 0,C 180,E1 7026.142,E2 7026.142} C_VEL
LIN {X 0,Y 138.747,Z 892.688,A -85,B 0,C 180,E1 7018.761,E2 7018.761} C_VEL
LIN {X 0,Y 138.652,Z 891.909,A -85,B 0,C 180,E1 7017.934,E2 7017.934} C_VEL
LIN {X 0,Y 139.357,Z 890.625,A -85,B 0,C 180,E1 7014.235,E2 7014.235} C_VEL
LIN {X 0,Y 139.949,Z 889.94,A -85,B 0,C 180,E1 7012.198,E2 7012.198} C_VEL
LIN {X 0,Y 141.861,Z 888.452,A -85,B 0,C 180,E1 7008.205,E2 7008.205} C_VEL
LIN {X 0,Y 151.117,Z 884.139,A -85,B 0,C 180,E1 6997.433,E2 6997.433} C_VEL
LIN {X 0,Y 161.731,Z 880.534,A -85,B 0,C 180,E1 6990.357,E2 6990.357} C_VEL
LIN {X 0,Y 176.432,Z 876.109,A -85,B 0,C 180,E1 6983.886,E2 6983.886} C_VEL
LIN {X 0,Y 187.683,Z 872.879,A -85,B 0,C 180,E1 6980.231,E2 6980.231} C_VEL
LIN {X 0,Y 175.991,Z 883.431,A -85,B 0,C 180,E1 6975.21,E2 6975.21} C_VEL
LIN {X 0,Y 165.356,Z 892.3,A -85,B 0,C 180,E1 6969.415,E2 6969.415} C_VEL
LIN {X 0,Y 155.917,Z 899.704,A -85,B 0,C 180,E1 6962.595,E2 6962.595} C_VEL
LIN {X 0,Y 148.567,Z 905.284,A -85,B 0,C 180,E1 6955.088,E2 6955.088} C_VEL
LIN {X 0,Y 143.438,Z 909.177,A -85,B 0,C 180,E1 6947.025,E2 6947.025} C_VEL
LIN {X 0,Y 140.551,Z 911.477,A -85,B 0,C 180,E1 6938.56,E2 6938.56} C_VEL
LIN {X 0,Y 139.664,Z 912.242,A -85,B 0,C 180,E1 6930,E2 6930} C_VEL
LIN {X 0,Y 140.511,Z 911.519,A -85,B 0,C 180,E1 6921.55,E2 6921.55} C_VEL
LIN {X 0,Y 143.212,Z 909.371,A -85,B 0,C 180,E1 6913.366,E2 6913.366} C_VEL
LIN {X 0,Y 148.213,Z 905.599,A -85,B 0,C 180,E1 6905.275,E2 6905.275} C_VEL
LIN {X 0,Y 155.445,Z 900.141,A -85,B 0,C 180,E1 6897.731,E2 6897.731} C_VEL
LIN {X 0,Y 164.776,Z 892.87,A -85,B 0,C 180,E1 6890.87,E2 6890.87} C_VEL
LIN {X 0,Y 175.515,Z 883.986,A -85,B 0,C 180,E1 6884.944,E2 6884.944} C_VEL
LIN {X 0,Y 186.777,Z 873.9,A -85,B 0,C 180,E1 6880.046,E2 6880.046} C_VEL
LIN {X 0,Y 198.583,Z 862.311,A -85,B 0,C 180,E1 6875.84,E2 6875.84} C_VEL
LIN {X 0,Y 210.497,Z 849.365,A -85,B 0,C 180,E1 6872.272,E2 6872.272} C_VEL
LIN {X 0,Y 222.278,Z 835.044,A -85,B 0,C 180,E1 6869.228,E2 6869.228} C_VEL
LIN {X 0,Y 233.356,Z 819.821,A -85,B 0,C 180,E1 6866.698,E2 6866.698} C_VEL
LIN {X 0,Y 243.96,Z 803.186,A -85,B 0,C 180,E1 6864.511,E2 6864.511} C_VEL
LIN {X 0,Y 253.795,Z 785.269,A -85,B 0,C 180,E1 6862.638,E2 6862.638} C_VEL
LIN {X 0,Y 262.516,Z 766.436,A -85,B 0,C 180,E1 6861.065,E2 6861.065} C_VEL
LIN {X 0,Y 270.115,Z 746.368,A -85,B 0,C 180,E1 6859.737,E2 6859.737} C_VEL
LIN {X 0,Y 276.439,Z 725.063,A -85,B 0,C 180,E1 6858.619,E2 6858.619} C_VEL
LIN {X 0,Y 286.245,Z 686.178,A -85,B 0,C 180,E1 6857.042,E2 6857.042} C_VEL
LIN {X 0,Y 295.072,Z 647.332,A -85,B 0,C 180,E1 6855.879,E2 6855.879} C_VEL
LIN {X 0,Y 303.348,Z 604.971,A -85,B 0,C 180,E1 6854.964,E2 6854.964} C_VEL
LIN {X 0,Y 309.935,Z 562.716,A -85,B 0,C 180,E1 6854.198,E2 6854.198} C_VEL
LIN {X 0,Y 316.767,Z 503.485,A -85,B 0,C 180,E1 6853.282,E2 6853.282} C_VEL
LIN {X 0,Y 318.692,Z 488.261,A -85,B 0,C 180,E1 6853.047,E2 6853.047} C_VEL
LIN {X 0,Y 319.062,Z 486.716,A -85,B 0,C 180,E1 6852.994,E2 6852.994} C_VEL
LIN {X 0,Y 318.382,Z 479.662,A -85,B 0,C 180,E1 6849.855,E2 6849.855} C_VEL
LIN {X 0,Y 318.091,Z 474.647,A -85,B 0,C 180,E1 6846.86,E2 6846.86} C_VEL
LIN {X 0,Y 318.171,Z 471.916,A -85,B 0,C 180,E1 6844.506,E2 6844.506} C_VEL
LIN {X 0,Y 318.595,Z 469.461,A -85,B 0,C 180,E1 6841.619,E2 6841.619} C_VEL
LIN {X 0,Y 319.79,Z 469.035,A -85,B 0,C 180,E1 6837.626,E2 6837.626} C_VEL
LIN {X 0,Y 319.391,Z 477.958,A -85,B 0,C 180,E1 6834.701,E2 6834.701} C_VEL
LIN {X 0,Y 319.36,Z 481.29,A -85,B 0,C 180,E1 6833.755,E2 6833.755} C_VEL
LIN {X 0,Y 308.857,Z 531.488,A -85,B 0,C 180,E1 6832.682,E2 6832.682} C_VEL
LIN {X 0,Y 304.602,Z 570.726,A -85,B 0,C 180,E1 6831.937,E2 6831.937} C_VEL
LIN {X 0,Y 303.585,Z 578.422,A -85,B 0,C 180,E1 6831.977,E2 6831.977} C_VEL
LIN {X 0,Y 299.983,Z 598.958,A -85,B 0,C 180,E1 6832.772,E2 6832.772} C_VEL
LIN {X 0,Y 298.908,Z 605.538,A -85,B 0,C 180,E1 6832.783,E2 6832.783} C_VEL
LIN {X 0,Y 292.126,Z 644.737,A -85,B 0,C 180,E1 6832.041,E2 6832.041} C_VEL
LIN {X 0,Y 283.674,Z 683.5,A -85,B 0,C 180,E1 6831.144,E2 6831.144} C_VEL
LIN {X 0,Y 274.58,Z 718.346,A -85,B 0,C 180,E1 6830.145,E2 6830.145} C_VEL
LIN {X 0,Y 265.214,Z 749.721,A -85,B 0,C 180,E1 6829.001,E2 6829.001} C_VEL
LIN {X 0,Y 256.749,Z 774.715,A -85,B 0,C 180,E1 6827.823,E2 6827.823} C_VEL
LIN {X 0,Y 248.354,Z 794.709,A -85,B 0,C 180,E1 6826.62,E2 6826.62} C_VEL
LIN {X 0,Y 238.929,Z 813.466,A -85,B 0,C 180,E1 6825.174,E2 6825.174} C_VEL
LIN {X 0,Y 227.892,Z 832.166,A -85,B 0,C 180,E1 6823.327,E2 6823.327} C_VEL
LIN {X 0,Y 215.73,Z 850.037,A -85,B 0,C 180,E1 6821,E2 6821} C_VEL
LIN {X 0,Y 203.452,Z 865.975,A -85,B 0,C 180,E1 6818.258,E2 6818.258} C_VEL
LIN {X 0,Y 190.921,Z 880.546,A -85,B 0,C 180,E1 6814.962,E2 6814.962} C_VEL
LIN {X 0,Y 177.634,Z 894.634,A -85,B 0,C 180,E1 6810.678,E2 6810.678} C_VEL
LIN {X 0,Y 165.007,Z 906.981,A -85,B 0,C 180,E1 6805.499,E2 6805.499} C_VEL
LIN {X 0,Y 153.681,Z 917.511,A -85,B 0,C 180,E1 6799.411,E2 6799.411} C_VEL
LIN {X 0,Y 143.666,Z 926.783,A -85,B 0,C 180,E1 6791.923,E2 6791.923} C_VEL
LIN {X 0,Y 136.167,Z 934.249,A -85,B 0,C 180,E1 6783.417,E2 6783.417} C_VEL
LIN {X 0,Y 131.636,Z 939.904,A -85,B 0,C 180,E1 6774.216,E2 6774.216} C_VEL
LIN {X 0,Y 130.073,Z 943.825,A -85,B 0,C 180,E1 6764.695,E2 6764.695} C_VEL
LIN {X 0,Y 130.754,Z 945.872,A -85,B 0,C 180,E1 6756.146,E2 6756.146} C_VEL
LIN {X 0,Y 131.553,Z 946.403,A -85,B 0,C 180,E1 6750.871,E2 6750.871} C_VEL
LIN {X 0,Y 131.255,Z 946.219,A -85,B 0,C 180,E1 6746.336,E2 6746.336} C_VEL
LIN {X 0,Y 130.432,Z 944.755,A -85,B 0,C 180,E1 6738.503,E2 6738.503} C_VEL
LIN {X 0,Y 131.622,Z 941.268,A -85,B 0,C 180,E1 6728.614,E2 6728.614} C_VEL
LIN {X 0,Y 136.128,Z 936.145,A -85,B 0,C 180,E1 6719.058,E2 6719.058} C_VEL
LIN {X 0,Y 150.072,Z 934.581,A -85,B 0,C 180,E1 6704.394,E2 6704.394} C_VEL
LIN {X 0,Y 163.874,Z 932.543,A -85,B 0,C 180,E1 6696.466,E2 6696.466} C_VEL
LIN {X 0,Y 150.837,Z 926.373,A -85,B 0,C 180,E1 6689.376,E2 6689.376} C_VEL
LIN {X 0,Y 141.01,Z 918.536,A -85,B 0,C 180,E1 6681.201,E2 6681.201} C_VEL
LIN {X 0,Y 134.919,Z 909.631,A -85,B 0,C 180,E1 6672.846,E2 6672.846} C_VEL
LIN {X 0,Y 131.698,Z 899.21,A -85,B 0,C 180,E1 6664.354,E2 6664.354} C_VEL
LIN {X 0,Y 131.396,Z 897.616,A -85,B 0,C 180,E1 6663.053,E2 6663.053} C_VEL
LIN {X 0,Y 131.291,Z 896.368,A -85,B 0,C 180,E1 6659.127,E2 6659.127} C_VEL
LIN {X 0,Y 131.636,Z 895.609,A -85,B 0,C 180,E1 6656.952,E2 6656.952} C_VEL
LIN {X 0,Y 133.054,Z 893.881,A -85,B 0,C 180,E1 6651.791,E2 6651.791} C_VEL
LIN {X 0,Y 145.133,Z 887.999,A -85,B 0,C 180,E1 6636.016,E2 6636.016} C_VEL
LIN {X 0,Y 160.953,Z 883.121,A -85,B 0,C 180,E1 6626.434,E2 6626.434} C_VEL
LIN {X 0,Y 177.556,Z 878.499,A -85,B 0,C 180,E1 6620.176,E2 6620.176} C_VEL
LIN {X 0,Y 165.266,Z 888.707,A -85,B 0,C 180,E1 6614.574,E2 6614.574} C_VEL
LIN {X 0,Y 154.247,Z 897.11,A -85,B 0,C 180,E1 6608.013,E2 6608.013} C_VEL
LIN {X 0,Y 145.127,Z 903.677,A -85,B 0,C 180,E1 6600.545,E2 6600.545} C_VEL
LIN {X 0,Y 138.174,Z 908.541,A -85,B 0,C 180,E1 6592.105,E2 6592.105} C_VEL
LIN {X 0,Y 133.91,Z 911.574,A -85,B 0,C 180,E1 6583.384,E2 6583.384} C_VEL
LIN {X 0,Y 131.939,Z 913.06,A -85,B 0,C 180,E1 6574.347,E2 6574.347} C_VEL
LIN {X 0,Y 131.929,Z 913.069,A -85,B 0,C 180,E1 6565.654,E2 6565.654} C_VEL
LIN {X 0,Y 133.738,Z 911.71,A -85,B 0,C 180,E1 6557.039,E2 6557.039} C_VEL
LIN {X 0,Y 137.866,Z 908.793,A -85,B 0,C 180,E1 6548.292,E2 6548.292} C_VEL
LIN {X 0,Y 144.406,Z 904.245,A -85,B 0,C 180,E1 6540.097,E2 6540.097} C_VEL
LIN {X 0,Y 153.219,Z 897.953,A -85,B 0,C 180,E1 6532.634,E2 6532.634} C_VEL
LIN {X 0,Y 163.489,Z 890.199,A -85,B 0,C 180,E1 6526.283,E2 6526.283} C_VEL
LIN {X 0,Y 174.695,Z 881.086,A -85,B 0,C 180,E1 6520.93,E2 6520.93} C_VEL
LIN {X 0,Y 186.416,Z 870.683,A -85,B 0,C 180,E1 6516.432,E2 6516.432} C_VEL
LIN {X 0,Y 199.022,Z 858.306,A -85,B 0,C 180,E1 6512.431,E2 6512.431} C_VEL
LIN {X 0,Y 211.613,Z 844.474,A -85,B 0,C 180,E1 6509.057,E2 6509.057} C_VEL
LIN {X 0,Y 223.463,Z 829.758,A -85,B 0,C 180,E1 6506.294,E2 6506.294} C_VEL
LIN {X 0,Y 234.704,Z 813.874,A -85,B 0,C 180,E1 6503.962,E2 6503.962} C_VEL
LIN {X 0,Y 245.275,Z 796.649,A -85,B 0,C 180,E1 6501.963,E2 6501.963} C_VEL
LIN {X 0,Y 254.773,Z 778.488,A -85,B 0,C 180,E1 6500.284,E2 6500.284} C_VEL
LIN {X 0,Y 263.118,Z 759.391,A -85,B 0,C 180,E1 6498.873,E2 6498.873} C_VEL
LIN {X 0,Y 270.288,Z 739.093,A -85,B 0,C 180,E1 6497.68,E2 6497.68} C_VEL
LIN {X 0,Y 279.287,Z 706.135,A -85,B 0,C 180,E1 6496.202,E2 6496.202} C_VEL
LIN {X 0,Y 288.343,Z 669.322,A -85,B 0,C 180,E1 6494.941,E2 6494.941} C_VEL
LIN {X 0,Y 296.706,Z 630.979,A -85,B 0,C 180,E1 6493.99,E2 6493.99} C_VEL
LIN {X 0,Y 304.282,Z 589.346,A -85,B 0,C 180,E1 6493.195,E2 6493.195} C_VEL
LIN {X 0,Y 310.403,Z 545.763,A -85,B 0,C 180,E1 6492.483,E2 6492.483} C_VEL
LIN {X 0,Y 316.559,Z 491.823,A -85,B 0,C 180,E1 6491.663,E2 6491.663} C_VEL
LIN {X 0,Y 316.136,Z 485.383,A -85,B 0,C 180,E1 6488.549,E2 6488.549} C_VEL
LIN {X 0,Y 316.087,Z 481.274,A -85,B 0,C 180,E1 6485.81,E2 6485.81} C_VEL
LIN {X 0,Y 316.278,Z 479.178,A -85,B 0,C 180,E1 6483.807,E2 6483.807} C_VEL
LIN {X 0,Y 316.762,Z 477.214,A -85,B 0,C 180,E1 6481.447,E2 6481.447} C_VEL
LIN {X 0,Y 317.777,Z 476.774,A -85,B 0,C 180,E1 6477.971,E2 6477.971} C_VEL
LIN {X 0,Y 317.328,Z 485.126,A -85,B 0,C 180,E1 6475.255,E2 6475.255} C_VEL
LIN {X 0,Y 317.251,Z 485.961,A -85,B 0,C 180,E1 6475.093,E2 6475.093} C_VEL
LIN {X 0,Y 308.165,Z 528.507,A -85,B 0,C 180,E1 6474.219,E2 6474.219} C_VEL
LIN {X 0,Y 300.294,Z 596.054,A -85,B 0,C 180,E1 6472.959,E2 6472.959} C_VEL
LIN {X 0,Y 298.908,Z 605.538,A -85,B 0,C 180,E1 6472.783,E2 6472.783} C_VEL
LIN {X 0,Y 297.623,Z 613.185,A -85,B 0,C 180,E1 6472.834,E2 6472.834} C_VEL
LIN {X 0,Y 293.15,Z 633.523,A -85,B 0,C 180,E1 6473.668,E2 6473.668} C_VEL
LIN {X 0,Y 291.743,Z 640.045,A -85,B 0,C 180,E1 6473.686,E2 6473.686} C_VEL
LIN {X 0,Y 283.564,Z 677.85,A -85,B 0,C 180,E1 6472.877,E2 6472.877} C_VEL
LIN {X 0,Y 274.126,Z 714.138,A -85,B 0,C 180,E1 6471.92,E2 6471.92} C_VEL
LIN {X 0,Y 264.128,Z 747.376,A -85,B 0,C 180,E1 6470.788,E2 6470.788} C_VEL
LIN {X 0,Y 255.598,Z 772.323,A -85,B 0,C 180,E1 6469.691,E2 6469.691} C_VEL
LIN {X 0,Y 247.216,Z 792.135,A -85,B 0,C 180,E1 6468.569,E2 6468.569} C_VEL
LIN {X 0,Y 237.839,Z 810.619,A -85,B 0,C 180,E1 6467.249,E2 6467.249} C_VEL
LIN {X 0,Y 227.114,Z 828.659,A -85,B 0,C 180,E1 6465.597,E2 6465.597} C_VEL
LIN {X 0,Y 215.477,Z 845.69,A -85,B 0,C 180,E1 6463.557,E2 6463.557} C_VEL
LIN {X 0,Y 202.861,Z 861.92,A -85,B 0,C 180,E1 6461.016,E2 6461.016} C_VEL
LIN {X 0,Y 189.092,Z 877.629,A -85,B 0,C 180,E1 6457.725,E2 6457.725} C_VEL
LIN {X 0,Y 175.969,Z 891.153,A -85,B 0,C 180,E1 6453.868,E2 6453.868} C_VEL
LIN {X 0,Y 163.071,Z 903.351,A -85,B 0,C 180,E1 6449.14,E2 6449.14} C_VEL
LIN {X 0,Y 150.851,Z 914.202,A -85,B 0,C 180,E1 6443.324,E2 6443.324} C_VEL
LIN {X 0,Y 139.642,Z 923.886,A -85,B 0,C 180,E1 6436.008,E2 6436.008} C_VEL
LIN {X 0,Y 130.601,Z 931.904,A -85,B 0,C 180,E1 6427.216,E2 6427.216} C_VEL
LIN {X 0,Y 124.836,Z 937.897,A -85,B 0,C 180,E1 6417.681,E2 6417.681} C_VEL
LIN {X 0,Y 122.274,Z 942.151,A -85,B 0,C 180,E1 6407.611,E2 6407.611} C_VEL
LIN {X 0,Y 122.512,Z 944.619,A -85,B 0,C 180,E1 6397.975,E2 6397.975} C_VEL
LIN {X 0,Y 123.554,Z 945.374,A -85,B 0,C 180,E1 6391.391,E2 6391.391} C_VEL
LIN {X 0,Y 123.482,Z 945.318,A -85,B 0,C 180,E1 6387.679,E2 6387.679} C_VEL
LIN {X 0,Y 122.538,Z 944.296,A -85,B 0,C 180,E1 6380.133,E2 6380.133} C_VEL
LIN {X 0,Y 123.22,Z 941.367,A -85,B 0,C 180,E1 6370.073,E2 6370.073} C_VEL
LIN {X 0,Y 127.422,Z 936.412,A -85,B 0,C 180,E1 6359.676,E2 6359.676} C_VEL
LIN {X 0,Y 130.796,Z 933.61,A -85,B 0,C 180,E1 6355.015,E2 6355.015} C_VEL
LIN {X 0,Y 146.55,Z 932.224,A -85,B 0,C 180,E1 6340.77,E2 6340.77} C_VEL
LIN {X 0,Y 153.997,Z 931.267,A -85,B 0,C 180,E1 6336.581,E2 6336.581} C_VEL
LIN {X 0,Y 140.918,Z 924.181,A -85,B 0,C 180,E1 6328.849,E2 6328.849} C_VEL
LIN {X 0,Y 131.806,Z 915.915,A -85,B 0,C 180,E1 6320.424,E2 6320.424} C_VEL
LIN {X 0,Y 126.086,Z 906.158,A -85,B 0,C 180,E1 6311.435,E2 6311.435} C_VEL
LIN {X 0,Y 124.965,Z 903.28,A -85,B 0,C 180,E1 6308.744,E2 6308.744} C_VEL
LIN {X 0,Y 124.169,Z 901.608,A -85,B 0,C 180,E1 6303.694,E2 6303.694} C_VEL
LIN {X 0,Y 124.649,Z 899.12,A -85,B 0,C 180,E1 6295.86,E2 6295.86} C_VEL
LIN {X 0,Y 126.324,Z 897.358,A -85,B 0,C 180,E1 6290.432,E2 6290.432} C_VEL
LIN {X 0,Y 143.508,Z 890.285,A -85,B 0,C 180,E1 6271.265,E2 6271.265} C_VEL
LIN {X 0,Y 163.76,Z 884.642,A -85,B 0,C 180,E1 6261.479,E2 6261.479} C_VEL
LIN {X 0,Y 167.509,Z 883.655,A -85,B 0,C 180,E1 6260.176,E2 6260.176} C_VEL
LIN {X 0,Y 155.027,Z 893.177,A -85,B 0,C 180,E1 6254.154,E2 6254.154} C_VEL
LIN {X 0,Y 144.113,Z 900.842,A -85,B 0,C 180,E1 6247.13,E2 6247.13} C_VEL
LIN {X 0,Y 134.985,Z 906.898,A -85,B 0,C 180,E1 6238.783,E2 6238.783} C_VEL
LIN {X 0,Y 128.518,Z 911.072,A -85,B 0,C 180,E1 6229.545,E2 6229.545} C_VEL
LIN {X 0,Y 124.863,Z 913.482,A -85,B 0,C 180,E1 6219.682,E2 6219.682} C_VEL
LIN {X 0,Y 123.789,Z 914.243,A -85,B 0,C 180,E1 6210,E2 6210} C_VEL
LIN {X 0,Y 124.741,Z 913.563,A -85,B 0,C 180,E1 6200.775,E2 6200.775} C_VEL
LIN {X 0,Y 128.027,Z 911.398,A -85,B 0,C 180,E1 6191.325,E2 6191.325} C_VEL
LIN {X 0,Y 133.884,Z 907.644,A -85,B 0,C 180,E1 6182.417,E2 6182.417} C_VEL
LIN {X 0,Y 142.191,Z 902.207,A -85,B 0,C 180,E1 6174.292,E2 6174.292} C_VEL
LIN {X 0,Y 152.27,Z 895.265,A -85,B 0,C 180,E1 6167.346,E2 6167.346} C_VEL
LIN {X 0,Y 163.846,Z 886.686,A -85,B 0,C 180,E1 6161.356,E2 6161.356} C_VEL
LIN {X 0,Y 176.249,Z 876.617,A -85,B 0,C 180,E1 6156.333,E2 6156.333} C_VEL
LIN {X 0,Y 188.963,Z 865.176,A -85,B 0,C 180,E1 6152.153,E2 6152.153} C_VEL
LIN {X 0,Y 201.681,Z 852.388,A -85,B 0,C 180,E1 6148.655,E2 6148.655} C_VEL
LIN {X 0,Y 214.17,Z 838.231,A -85,B 0,C 180,E1 6145.703,E2 6145.703} C_VEL
LIN {X 0,Y 226.259,Z 822.637,A -85,B 0,C 180,E1 6143.191,E2 6143.191} C_VEL
LIN {X 0,Y 237.401,Z 806.096,A -85,B 0,C 180,E1 6141.106,E2 6141.106} C_VEL
LIN {X 0,Y 247.9,Z 787.962,A -85,B 0,C 180,E1 6139.296,E2 6139.296} C_VEL
LIN {X 0,Y 257.242,Z 768.611,A -85,B 0,C 180,E1 6137.767,E2 6137.767} C_VEL
LIN {X 0,Y 264.943,Z 749.12,A -85,B 0,C 180,E1 6136.546,E2 6136.546} C_VEL
LIN {X 0,Y 271.413,Z 728.406,A -85,B 0,C 180,E1 6135.507,E2 6135.507} C_VEL
LIN {X 0,Y 281.158,Z 691.859,A -85,B 0,C 180,E1 6134.073,E2 6134.073} C_VEL
LIN {X 0,Y 289.738,Z 656.317,A -85,B 0,C 180,E1 6133.027,E2 6133.027} C_VEL
LIN {X 0,Y 297.75,Z 618.076,A -85,B 0,C 180,E1 6132.22,E2 6132.22} C_VEL
LIN {X 0,Y 304.748,Z 576.937,A -85,B 0,C 180,E1 6131.503,E2 6131.503} C_VEL
LIN {X 0,Y 310.385,Z 533.116,A -85,B 0,C 180,E1 6130.843,E2 6130.843} C_VEL
LIN {X 0,Y 314.378,Z 497.094,A -85,B 0,C 180,E1 6130.311,E2 6130.311} C_VEL
LIN {X 0,Y 314.045,Z 491.397,A -85,B 0,C 180,E1 6127.317,E2 6127.317} C_VEL
LIN {X 0,Y 314.25,Z 487.496,A -85,B 0,C 180,E1 6124.38,E2 6124.38} C_VEL
LIN {X 0,Y 314.958,Z 484.973,A -85,B 0,C 180,E1 6121.273,E2 6121.273} C_VEL
LIN {X 0,Y 315.776,Z 484.695,A -85,B 0,C 180,E1 6118.276,E2 6118.276} C_VEL
LIN {X 0,Y 315.345,Z 490.279,A -85,B 0,C 180,E1 6116.452,E2 6116.452} C_VEL
LIN {X 0,Y 307.684,Z 525.631,A -85,B 0,C 180,E1 6115.759,E2 6115.759} C_VEL
LIN {X 0,Y 299.585,Z 593.552,A -85,B 0,C 180,E1 6114.522,E2 6114.522} C_VEL
LIN {X 0,Y 293.231,Z 632.503,A -85,B 0,C 180,E1 6113.825,E2 6113.825} C_VEL
LIN {X 0,Y 291.743,Z 640.045,A -85,B 0,C 180,E1 6113.686,E2 6113.686} C_VEL
LIN {X 0,Y 290.098,Z 647.63,A -85,B 0,C 180,E1 6113.746,E2 6113.746} C_VEL
LIN {X 0,Y 284.562,Z 668.867,A -85,B 0,C 180,E1 6114.587,E2 6114.587} C_VEL
LIN {X 0,Y 283.18,Z 674.24,A -85,B 0,C 180,E1 6114.562,E2 6114.562} C_VEL
LIN {X 0,Y 273.552,Z 711.211,A -85,B 0,C 180,E1 6113.654,E2 6113.654} C_VEL
LIN {X 0,Y 262.941,Z 746.099,A -85,B 0,C 180,E1 6112.55,E2 6112.55} C_VEL
LIN {X 0,Y 254.254,Z 771.078,A -85,B 0,C 180,E1 6111.517,E2 6111.517} C_VEL
LIN {X 0,Y 245.865,Z 790.576,A -85,B 0,C 180,E1 6110.472,E2 6110.472} C_VEL
LIN {X 0,Y 236.148,Z 809.356,A -85,B 0,C 180,E1 6109.212,E2 6109.212} C_VEL
LIN {X 0,Y 225.191,Z 827.407,A -85,B 0,C 180,E1 6107.645,E2 6107.645} C_VEL
LIN {X 0,Y 213.547,Z 844.088,A -85,B 0,C 180,E1 6105.751,E2 6105.751} C_VEL
LIN {X 0,Y 200.977,Z 859.884,A -85,B 0,C 180,E1 6103.428,E2 6103.428} C_VEL
LIN {X 0,Y 186.892,Z 875.571,A -85,B 0,C 180,E1 6100.325,E2 6100.325} C_VEL
LIN {X 0,Y 172.606,Z 889.815,A -85,B 0,C 180,E1 6096.44,E2 6096.44} C_VEL
LIN {X 0,Y 158.904,Z 902.205,A -85,B 0,C 180,E1 6091.755,E2 6091.755} C_VEL
LIN {X 0,Y 145.971,Z 913.076,A -85,B 0,C 180,E1 6085.98,E2 6085.98} C_VEL
LIN {X 0,Y 134.202,Z 922.546,A -85,B 0,C 180,E1 6078.808,E2 6078.808} C_VEL
LIN {X 0,Y 124.409,Z 930.496,A -85,B 0,C 180,E1 6070.013,E2 6070.013} C_VEL
LIN {X 0,Y 117.675,Z 936.658,A -85,B 0,C 180,E1 6059.922,E2 6059.922} C_VEL
LIN {X 0,Y 114.432,Z 941.1,A -85,B 0,C 180,E1 6048.862,E2 6048.862} C_VEL
LIN {X 0,Y 114.474,Z 943.592,A -85,B 0,C 180,E1 6038.539,E2 6038.539} C_VEL
LIN {X 0,Y 115.589,Z 944.369,A -85,B 0,C 180,E1 6031.487,E2 6031.487} C_VEL
LIN {X 0,Y 115.509,Z 944.312,A -85,B 0,C 180,E1 6027.519,E2 6027.519} C_VEL
LIN {X 0,Y 114.53,Z 943.156,A -85,B 0,C 180,E1 6018.926,E2 6018.926} C_VEL
LIN {X 0,Y 115.655,Z 940.131,A -85,B 0,C 180,E1 6008.176,E2 6008.176} C_VEL
LIN {X 0,Y 120.599,Z 935.16,A -85,B 0,C 180,E1 5997.39,E2 5997.39} C_VEL
LIN {X 0,Y 126.155,Z 930.988,A -85,B 0,C 180,E1 5990.648,E2 5990.648} C_VEL
LIN {X 0,Y 143.23,Z 929.701,A -85,B 0,C 180,E1 5977.265,E2 5977.265} C_VEL
LIN {X 0,Y 144.045,Z 929.534,A -85,B 0,C 180,E1 5976.653,E2 5976.653} C_VEL
LIN {X 0,Y 131.517,Z 921.923,A -85,B 0,C 180,E1 5968.618,E2 5968.618} C_VEL
LIN {X 0,Y 122.649,Z 912.864,A -85,B 0,C 180,E1 5959.527,E2 5959.527} C_VEL
LIN {X 0,Y 119.971,Z 908.753,A -85,B 0,C 180,E1 5955.468,E2 5955.468} C_VEL
LIN {X 0,Y 117.846,Z 906.924,A -85,B 0,C 180,E1 5949.77,E2 5949.77} C_VEL
LIN {X 0,Y 116.77,Z 904.113,A -85,B 0,C 180,E1 5940.491,E2 5940.491} C_VEL
LIN {X 0,Y 117.529,Z 902.473,A -85,B 0,C 180,E1 5935.12,E2 5935.12} C_VEL
LIN {X 0,Y 137.218,Z 893.895,A -85,B 0,C 180,E1 5909.815,E2 5909.815} C_VEL
LIN {X 0,Y 157.255,Z 888.639,A -85,B 0,C 180,E1 5900.105,E2 5900.105} C_VEL
LIN {X 0,Y 144.759,Z 897.353,A -85,B 0,C 180,E1 5893.688,E2 5893.688} C_VEL
LIN {X 0,Y 133.967,Z 904.276,A -85,B 0,C 180,E1 5886.131,E2 5886.131} C_VEL
LIN {X 0,Y 125.152,Z 909.614,A -85,B 0,C 180,E1 5877.091,E2 5877.091} C_VEL
LIN {X 0,Y 119.428,Z 912.999,A -85,B 0,C 180,E1 5867.542,E2 5867.542} C_VEL
LIN {X 0,Y 116.437,Z 914.813,A -85,B 0,C 180,E1 5857.401,E2 5857.401} C_VEL
LIN {X 0,Y 115.901,Z 915.159,A -85,B 0,C 180,E1 5847.528,E2 5847.528} C_VEL
LIN {X 0,Y 117.515,Z 914.184,A -85,B 0,C 180,E1 5837.719,E2 5837.719} C_VEL
LIN {X 0,Y 121.768,Z 911.67,A -85,B 0,C 180,E1 5827.807,E2 5827.807} C_VEL
LIN {X 0,Y 128.759,Z 907.546,A -85,B 0,C 180,E1 5818.648,E2 5818.648} C_VEL
LIN {X 0,Y 138.261,Z 901.699,A -85,B 0,C 180,E1 5810.476,E2 5810.476} C_VEL
LIN {X 0,Y 149.737,Z 894.118,A -85,B 0,C 180,E1 5803.456,E2 5803.456} C_VEL
LIN {X 0,Y 161.984,Z 885.293,A -85,B 0,C 180,E1 5797.804,E2 5797.804} C_VEL
LIN {X 0,Y 175.23,Z 874.715,A -85,B 0,C 180,E1 5792.986,E2 5792.986} C_VEL
LIN {X 0,Y 188.65,Z 862.724,A -85,B 0,C 180,E1 5789.01,E2 5789.01} C_VEL
LIN {X 0,Y 201.959,Z 849.303,A -85,B 0,C 180,E1 5785.701,E2 5785.701} C_VEL
LIN {X 0,Y 214.942,Z 834.399,A -85,B 0,C 180,E1 5782.916,E2 5782.916} C_VEL
LIN {X 0,Y 226.972,Z 818.579,A -85,B 0,C 180,E1 5780.636,E2 5780.636} C_VEL
LIN {X 0,Y 238.077,Z 801.689,A -85,B 0,C 180,E1 5778.725,E2 5778.725} C_VEL
LIN {X 0,Y 247.55,Z 784.883,A -85,B 0,C 180,E1 5777.204,E2 5777.204} C_VEL
LIN {X 0,Y 256.113,Z 766.908,A -85,B 0,C 180,E1 5775.887,E2 5775.887} C_VEL
LIN {X 0,Y 263.228,Z 748.875,A -85,B 0,C 180,E1 5774.82,E2 5774.82} C_VEL
LIN {X 0,Y 269.781,Z 728.009,A -85,B 0,C 180,E1 5773.82,E2 5773.82} C_VEL
LIN {X 0,Y 279.027,Z 694.221,A -85,B 0,C 180,E1 5772.535,E2 5772.535} C_VEL
LIN {X 0,Y 287.478,Z 660.233,A -85,B 0,C 180,E1 5771.554,E2 5771.554} C_VEL
LIN {X 0,Y 295.644,Z 622.289,A -85,B 0,C 180,E1 5770.77,E2 5770.77} C_VEL
LIN {X 0,Y 302.903,Z 580.645,A -85,B 0,C 180,E1 5770.07,E2 5770.07} C_VEL
LIN {X 0,Y 308.599,Z 537.418,A -85,B 0,C 180,E1 5769.44,E2 5769.44} C_VEL
LIN {X 0,Y 312.519,Z 502.545,A -85,B 0,C 180,E1 5768.927,E2 5768.927} C_VEL
LIN {X 0,Y 312.032,Z 498.801,A -85,B 0,C 180,E1 5766.902,E2 5766.902} C_VEL
LIN {X 0,Y 312.365,Z 495.078,A -85,B 0,C 180,E1 5764.038,E2 5764.038} C_VEL
LIN {X 0,Y 313.051,Z 492.707,A -85,B 0,C 180,E1 5761.098,E2 5761.098} C_VEL
LIN {X 0,Y 313.821,Z 492.476,A -85,B 0,C 180,E1 5758.631,E2 5758.631} C_VEL
LIN {X 0,Y 313.536,Z 495.061,A -85,B 0,C 180,E1 5757.82,E2 5757.82} C_VEL
LIN {X 0,Y 307.401,Z 522.954,A -85,B 0,C 180,E1 5757.299,E2 5757.299} C_VEL
LIN {X 0,Y 299.158,Z 590.648,A -85,B 0,C 180,E1 5756.104,E2 5756.104} C_VEL
LIN {X 0,Y 292.682,Z 629.917,A -85,B 0,C 180,E1 5755.425,E2 5755.425} C_VEL
LIN {X 0,Y 284.385,Z 669.361,A -85,B 0,C 180,E1 5754.671,E2 5754.671} C_VEL
LIN {X 0,Y 283.18,Z 674.24,A -85,B 0,C 180,E1 5754.562,E2 5754.562} C_VEL
LIN {X 0,Y 281.187,Z 681.753,A -85,B 0,C 180,E1 5754.599,E2 5754.599} C_VEL
LIN {X 0,Y 275.194,Z 701.752,A -85,B 0,C 180,E1 5755.414,E2 5755.414} C_VEL
LIN {X 0,Y 273.269,Z 708.115,A -85,B 0,C 180,E1 5755.397,E2 5755.397} C_VEL
LIN {X 0,Y 262.244,Z 744.106,A -85,B 0,C 180,E1 5754.353,E2 5754.353} C_VEL
LIN {X 0,Y 253.647,Z 768.686,A -85,B 0,C 180,E1 5753.412,E2 5753.412} C_VEL
LIN {X 0,Y 245.11,Z 788.404,A -85,B 0,C 180,E1 5752.429,E2 5752.429} C_VEL
LIN {X 0,Y 235.208,Z 807.344,A -85,B 0,C 180,E1 5751.256,E2 5751.256} C_VEL
LIN {X 0,Y 223.563,Z 826.196,A -85,B 0,C 180,E1 5749.721,E2 5749.721} C_VEL
LIN {X 0,Y 211.318,Z 843.293,A -85,B 0,C 180,E1 5747.886,E2 5747.886} C_VEL
LIN {X 0,Y 197.751,Z 859.805,A -85,B 0,C 180,E1 5745.557,E2 5745.557} C_VEL
LIN {X 0,Y 184.234,Z 874.362,A -85,B 0,C 180,E1 5742.785,E2 5742.785} C_VEL
LIN {X 0,Y 170.038,Z 888.064,A -85,B 0,C 180,E1 5739.225,E2 5739.225} C_VEL
LIN {X 0,Y 155.84,Z 900.418,A -85,B 0,C 180,E1 5734.779,E2 5734.779} C_VEL
LIN {X 0,Y 141.908,Z 911.565,A -85,B 0,C 180,E1 5729.045,E2 5729.045} C_VEL
LIN {X 0,Y 128.724,Z 921.492,A -85,B 0,C 180,E1 5721.58,E2 5721.58} C_VEL
LIN {X 0,Y 117.954,Z 929.505,A -85,B 0,C 180,E1 5712.481,E2 5712.481} C_VEL
LIN {X 0,Y 110.325,Z 935.758,A -85,B 0,C 180,E1 5701.712,E2 5701.712} C_VEL
LIN {X 0,Y 106.56,Z 940.214,A -85,B 0,C 180,E1 5689.743,E2 5689.743} C_VEL
LIN {X 0,Y 106.497,Z 942.645,A -85,B 0,C 180,E1 5678.639,E2 5678.639} C_VEL
LIN {X 0,Y 107.684,Z 943.393,A -85,B 0,C 180,E1 5671.064,E2 5671.064} C_VEL
LIN {X 0,Y 107.523,Z 943.304,A -85,B 0,C 180,E1 5667.335,E2 5667.335} C_VEL
LIN {X 0,Y 106.555,Z 942.128,A -85,B 0,C 180,E1 5658.086,E2 5658.086} C_VEL
LIN {X 0,Y 108.075,Z 939.083,A -85,B 0,C 180,E1 5646.557,E2 5646.557} C_VEL
LIN {X 0,Y 113.688,Z 934.082,A -85,B 0,C 180,E1 5635.132,E2 5635.132} C_VEL
LIN {X 0,Y 122.097,Z 928.266,A -85,B 0,C 180,E1 5626.211,E2 5626.211} C_VEL
LIN {X 0,Y 134.399,Z 927.526,A -85,B 0,C 180,E1 5616.881,E2 5616.881} C_VEL
LIN {X 0,Y 122.146,Z 919.286,A -85,B 0,C 180,E1 5608.346,E2 5608.346} C_VEL
LIN {X 0,Y 117.025,Z 914.146,A -85,B 0,C 180,E1 5603.144,E2 5603.144} C_VEL
LIN {X 0,Y 113.073,Z 912.173,A -85,B 0,C 180,E1 5596.967,E2 5596.967} C_VEL
LIN {X 0,Y 109.453,Z 907.385,A -85,B 0,C 180,E1 5580.523,E2 5580.523} C_VEL
LIN {X 0,Y 112.67,Z 903.773,A -85,B 0,C 180,E1 5567.702,E2 5567.702} C_VEL
LIN {X 0,Y 132.126,Z 896.959,A -85,B 0,C 180,E1 5547.499,E2 5547.499} C_VEL
LIN {X 0,Y 147.028,Z 893.272,A -85,B 0,C 180,E1 5540.066,E2 5540.066} C_VEL
LIN {X 0,Y 134.467,Z 901.254,A -85,B 0,C 180,E1 5533.166,E2 5533.166} C_VEL
LIN {X 0,Y 123.374,Z 907.709,A -85,B 0,C 180,E1 5524.564,E2 5524.564} C_VEL
LIN {X 0,Y 115.071,Z 912.271,A -85,B 0,C 180,E1 5514.651,E2 5514.651} C_VEL
LIN {X 0,Y 109.933,Z 915.057,A -85,B 0,C 180,E1 5503.679,E2 5503.679} C_VEL
LIN {X 0,Y 107.974,Z 916.152,A -85,B 0,C 180,E1 5492.654,E2 5492.654} C_VEL
LIN {X 0,Y 108.551,Z 915.84,A -85,B 0,C 180,E1 5482.058,E2 5482.058} C_VEL
LIN {X 0,Y 111.827,Z 914.064,A -85,B 0,C 180,E1 5471.223,E2 5471.223} C_VEL
LIN {X 0,Y 118.054,Z 910.725,A -85,B 0,C 180,E1 5461.133,E2 5461.133} C_VEL
LIN {X 0,Y 127.045,Z 905.724,A -85,B 0,C 180,E1 5452.129,E2 5452.129} C_VEL
LIN {X 0,Y 137.834,Z 899.315,A -85,B 0,C 180,E1 5444.69,E2 5444.69} C_VEL
LIN {X 0,Y 150.392,Z 891.155,A -85,B 0,C 180,E1 5438.323,E2 5438.323} C_VEL
LIN {X 0,Y 163.633,Z 881.615,A -85,B 0,C 180,E1 5433.16,E2 5433.16} C_VEL
LIN {X 0,Y 177.108,Z 870.743,A -85,B 0,C 180,E1 5428.947,E2 5428.947} C_VEL
LIN {X 0,Y 190.507,Z 858.582,A -85,B 0,C 180,E1 5425.478,E2 5425.478} C_VEL
LIN {X 0,Y 203.6,Z 845.135,A -85,B 0,C 180,E1 5422.59,E2 5422.59} C_VEL
LIN {X 0,Y 216.219,Z 830.357,A -85,B 0,C 180,E1 5420.156,E2 5420.156} C_VEL
LIN {X 0,Y 228.251,Z 814.145,A -85,B 0,C 180,E1 5418.084,E2 5418.084} C_VEL
LIN {X 0,Y 238.722,Z 797.816,A -85,B 0,C 180,E1 5416.43,E2 5416.43} C_VEL
LIN {X 0,Y 248.421,Z 780.045,A -85,B 0,C 180,E1 5414.985,E2 5414.985} C_VEL
LIN {X 0,Y 256.415,Z 762.648,A -85,B 0,C 180,E1 5413.839,E2 5413.839} C_VEL
LIN {X 0,Y 263.544,Z 743.638,A -85,B 0,C 180,E1 5412.823,E2 5412.823} C_VEL
LIN {X 0,Y 273.408,Z 710.345,A -85,B 0,C 180,E1 5411.446,E2 5411.446} C_VEL
LIN {X 0,Y 282.511,Z 675.791,A -85,B 0,C 180,E1 5410.359,E2 5410.359} C_VEL
LIN {X 0,Y 290.897,Z 639.692,A -85,B 0,C 180,E1 5409.539,E2 5409.539} C_VEL
LIN {X 0,Y 298.304,Z 601.913,A -85,B 0,C 180,E1 5408.894,E2 5408.894} C_VEL
LIN {X 0,Y 304.521,Z 561.656,A -85,B 0,C 180,E1 5408.293,E2 5408.293} C_VEL
LIN {X 0,Y 310.827,Z 508.179,A -85,B 0,C 180,E1 5407.533,E2 5407.533} C_VEL
LIN {X 0,Y 310.206,Z 504.294,A -85,B 0,C 180,E1 5405.124,E2 5405.124} C_VEL
LIN {X 0,Y 310.624,Z 502.045,A -85,B 0,C 180,E1 5402.952,E2 5402.952} C_VEL
LIN {X 0,Y 311.19,Z 500.451,A -85,B 0,C 180,E1 5400.921,E2 5400.921} C_VEL
LIN {X 0,Y 311.684,Z 500.279,A -85,B 0,C 180,E1 5399.193,E2 5399.193} C_VEL
LIN {X 0,Y 307.357,Z 520.155,A -85,B 0,C 180,E1 5398.841,E2 5398.841} C_VEL
LIN {X 0,Y 298.937,Z 587.892,A -85,B 0,C 180,E1 5397.686,E2 5397.686} C_VEL
LIN {X 0,Y 292.33,Z 627.482,A -85,B 0,C 180,E1 5397.025,E2 5397.025} C_VEL
LIN {X 0,Y 283.931,Z 667.082,A -85,B 0,C 180,E1 5396.323,E2 5396.323} C_VEL
LIN {X 0,Y 273.634,Z 706.852,A -85,B 0,C 180,E1 5395.429,E2 5395.429} C_VEL
LIN {X 0,Y 273.269,Z 708.115,A -85,B 0,C 180,E1 5395.397,E2 5395.397} C_VEL
LIN {X 0,Y 270.95,Z 715.525,A -85,B 0,C 180,E1 5395.402,E2 5395.402} C_VEL
LIN {X 0,Y 264.169,Z 735.309,A -85,B 0,C 180,E1 5396.207,E2 5396.207} C_VEL
LIN {X 0,Y 261.988,Z 741.591,A -85,B 0,C 180,E1 5396.18,E2 5396.18} C_VEL
LIN {X 0,Y 253.319,Z 766.281,A -85,B 0,C 180,E1 5395.313,E2 5395.313} C_VEL
LIN {X 0,Y 244.331,Z 786.818,A -85,B 0,C 180,E1 5394.364,E2 5394.364} C_VEL
LIN {X 0,Y 234.279,Z 805.781,A -85,B 0,C 180,E1 5393.279,E2 5393.279} C_VEL
LIN {X 0,Y 222.708,Z 824.293,A -85,B 0,C 180,E1 5391.881,E2 5391.881} C_VEL
LIN {X 0,Y 210.064,Z 841.669,A -85,B 0,C 180,E1 5390.165,E2 5390.165} C_VEL
LIN {X 0,Y 196.263,Z 858.133,A -85,B 0,C 180,E1 5388.006,E2 5388.006} C_VEL
LIN {X 0,Y 181.928,Z 873.186,A -85,B 0,C 180,E1 5385.309,E2 5385.309} C_VEL
LIN {X 0,Y 167.238,Z 886.889,A -85,B 0,C 180,E1 5381.922,E2 5381.922} C_VEL
LIN {X 0,Y 152.362,Z 899.309,A -85,B 0,C 180,E1 5377.627,E2 5377.627} C_VEL
LIN {X 0,Y 137.965,Z 910.277,A -85,B 0,C 180,E1 5372.151,E2 5372.151} C_VEL
LIN {X 0,Y 124.37,Z 919.877,A -85,B 0,C 180,E1 5365.089,E2 5365.089} C_VEL
LIN {X 0,Y 112.547,Z 927.982,A -85,B 0,C 180,E1 5356.023,E2 5356.023} C_VEL
LIN {X 0,Y 103.618,Z 934.442,A -85,B 0,C 180,E1 5344.703,E2 5344.703} C_VEL
LIN {X 0,Y 99.045,Z 938.841,A -85,B 0,C 180,E1 5332.558,E2 5332.558} C_VEL
LIN {X 0,Y 98.366,Z 941.455,A -85,B 0,C 180,E1 5320.542,E2 5320.542} C_VEL
LIN {X 0,Y 99.632,Z 942.357,A -85,B 0,C 180,E1 5311.725,E2 5311.725} C_VEL
LIN {X 0,Y 99.687,Z 942.359,A -85,B 0,C 180,E1 5308.275,E2 5308.275} C_VEL
LIN {X 0,Y 98.619,Z 941.398,A -85,B 0,C 180,E1 5298.893,E2 5298.893} C_VEL
LIN {X 0,Y 100.203,Z 938.422,A -85,B 0,C 180,E1 5285.85,E2 5285.85} C_VEL
LIN {X 0,Y 106.237,Z 933.564,A -85,B 0,C 180,E1 5273.633,E2 5273.633} C_VEL
LIN {X 0,Y 116.506,Z 926.832,A -85,B 0,C 180,E1 5263.155,E2 5263.155} C_VEL
LIN {X 0,Y 119.403,Z 925.309,A -85,B 0,C 180,E1 5261.091,E2 5261.091} C_VEL
LIN {X 0,Y 124.749,Z 925.094,A -85,B 0,C 180,E1 5257.105,E2 5257.105} C_VEL
LIN {X 0,Y 116.212,Z 919.228,A -85,B 0,C 180,E1 5251.081,E2 5251.081} C_VEL
LIN {X 0,Y 105.712,Z 915.062,A -85,B 0,C 180,E1 5237.618,E2 5237.618} C_VEL
LIN {X 0,Y 102.911,Z 908.863,A -85,B 0,C 180,E1 5214.424,E2 5214.424} C_VEL
LIN {X 0,Y 125.546,Z 900.271,A -85,B 0,C 180,E1 5185.924,E2 5185.924} C_VEL
LIN {X 0,Y 136.876,Z 897.562,A -85,B 0,C 180,E1 5180.089,E2 5180.089} C_VEL
LIN {X 0,Y 124.152,Z 904.891,A -85,B 0,C 180,E1 5172.573,E2 5172.573} C_VEL
LIN {X 0,Y 113.258,Z 910.617,A -85,B 0,C 180,E1 5163.187,E2 5163.187} C_VEL
LIN {X 0,Y 105.415,Z 914.504,A -85,B 0,C 180,E1 5152.298,E2 5152.298} C_VEL
LIN {X 0,Y 101.161,Z 916.605,A -85,B 0,C 180,E1 5140.825,E2 5140.825} C_VEL
LIN {X 0,Y 99.972,Z 917.237,A -85,B 0,C 180,E1 5129.427,E2 5129.427} C_VEL
LIN {X 0,Y 101.413,Z 916.524,A -85,B 0,C 180,E1 5118.051,E2 5118.051} C_VEL
LIN {X 0,Y 106.246,Z 914.18,A -85,B 0,C 180,E1 5106.129,E2 5106.129} C_VEL
LIN {X 0,Y 114.517,Z 910.086,A -85,B 0,C 180,E1 5095.421,E2 5095.421} C_VEL
LIN {X 0,Y 125.775,Z 904.102,A -85,B 0,C 180,E1 5086.241,E2 5086.241} C_VEL
LIN {X 0,Y 138.765,Z 896.517,A -85,B 0,C 180,E1 5078.904,E2 5078.904} C_VEL
LIN {X 0,Y 152.72,Z 887.421,A -85,B 0,C 180,E1 5073.066,E2 5073.066} C_VEL
LIN {X 0,Y 167.084,Z 876.867,A -85,B 0,C 180,E1 5068.394,E2 5068.394} C_VEL
LIN {X 0,Y 181.46,Z 864.89,A -85,B 0,C 180,E1 5064.606,E2 5064.606} C_VEL
LIN {X 0,Y 195.585,Z 851.485,A -85,B 0,C 180,E1 5061.497,E2 5061.497} C_VEL
LIN {X 0,Y 208.601,Z 837.38,A -85,B 0,C 180,E1 5059.023,E2 5059.023} C_VEL
LIN {X 0,Y 221.053,Z 821.901,A -85,B 0,C 180,E1 5056.927,E2 5056.927} C_VEL
LIN {X 0,Y 232.13,Z 806.011,A -85,B 0,C 180,E1 5055.232,E2 5055.232} C_VEL
LIN {X 0,Y 241.983,Z 789.593,A -85,B 0,C 180,E1 5053.824,E2 5053.824} C_VEL
LIN {X 0,Y 250.51,Z 772.939,A -85,B 0,C 180,E1 5052.657,E2 5052.657} C_VEL
LIN {X 0,Y 258.342,Z 754.518,A -85,B 0,C 180,E1 5051.611,E2 5051.611} C_VEL
LIN {X 0,Y 264.963,Z 735.092,A -85,B 0,C 180,E1 5050.711,E2 5050.711} C_VEL
LIN {X 0,Y 274.717,Z 701.51,A -85,B 0,C 180,E1 5049.474,E2 5049.474} C_VEL
LIN {X 0,Y 283.63,Z 667.686,A -85,B 0,C 180,E1 5048.541,E2 5048.541} C_VEL
LIN {X 0,Y 292.295,Z 629.173,A -85,B 0,C 180,E1 5047.787,E2 5047.787} C_VEL
LIN {X 0,Y 299.95,Z 586.992,A -85,B 0,C 180,E1 5047.141,E2 5047.141} C_VEL
LIN {X 0,Y 305.774,Z 544.445,A -85,B 0,C 180,E1 5046.569,E2 5046.569} C_VEL
LIN {X 0,Y 309.314,Z 514.061,A -85,B 0,C 180,E1 5046.17,E2 5046.17} C_VEL
LIN {X 0,Y 308.742,Z 510.419,A -85,B 0,C 180,E1 5043.528,E2 5043.528} C_VEL
LIN {X 0,Y 309.391,Z 508.21,A -85,B 0,C 180,E1 5040.741,E2 5040.741} C_VEL
LIN {X 0,Y 309.404,Z 508.336,A -85,B 0,C 180,E1 5040.533,E2 5040.533} C_VEL
LIN {X 0,Y 307.496,Z 517.68,A -85,B 0,C 180,E1 5040.378,E2 5040.378} C_VEL
LIN {X 0,Y 298.935,Z 585.198,A -85,B 0,C 180,E1 5039.268,E2 5039.268} C_VEL
LIN {X 0,Y 292.214,Z 625.014,A -85,B 0,C 180,E1 5038.629,E2 5038.629} C_VEL
LIN {X 0,Y 283.724,Z 664.757,A -85,B 0,C 180,E1 5037.98,E2 5037.98} C_VEL
LIN {X 0,Y 273.246,Z 704.978,A -85,B 0,C 180,E1 5037.145,E2 5037.145} C_VEL
LIN {X 0,Y 261.988,Z 741.591,A -85,B 0,C 180,E1 5036.18,E2 5036.18} C_VEL
LIN {X 0,Y 259.38,Z 748.911,A -85,B 0,C 180,E1 5036.159,E2 5036.159} C_VEL
LIN {X 0,Y 252.021,Z 767.378,A -85,B 0,C 180,E1 5036.853,E2 5036.853} C_VEL
LIN {X 0,Y 248.861,Z 774.442,A -85,B 0,C 180,E1 5036.794,E2 5036.794} C_VEL
LIN {X 0,Y 239.587,Z 793.606,A -85,B 0,C 180,E1 5035.898,E2 5035.898} C_VEL
LIN {X 0,Y 228.912,Z 812.088,A -85,B 0,C 180,E1 5034.813,E2 5034.813} C_VEL
LIN {X 0,Y 216.891,Z 829.847,A -85,B 0,C 180,E1 5033.451,E2 5033.451} C_VEL
LIN {X 0,Y 203.66,Z 846.745,A -85,B 0,C 180,E1 5031.72,E2 5031.72} C_VEL
LIN {X 0,Y 189.138,Z 862.871,A -85,B 0,C 180,E1 5029.513,E2 5029.513} C_VEL
LIN {X 0,Y 173.667,Z 877.908,A -85,B 0,C 180,E1 5026.66,E2 5026.66} C_VEL
LIN {X 0,Y 157.883,Z 891.47,A -85,B 0,C 180,E1 5022.999,E2 5022.999} C_VEL
LIN {X 0,Y 142.882,Z 902.971,A -85,B 0,C 180,E1 5018.549,E2 5018.549} C_VEL
LIN {X 0,Y 128.217,Z 913.193,A -85,B 0,C 180,E1 5012.75,E2 5012.75} C_VEL
LIN {X 0,Y 114.514,Z 922.062,A -85,B 0,C 180,E1 5005.161,E2 5005.161} C_VEL
LIN {X 0,Y 102.767,Z 929.47,A -85,B 0,C 180,E1 4995.256,E2 4995.256} C_VEL
LIN {X 0,Y 94.278,Z 935.285,A -85,B 0,C 180,E1 4982.744,E2 4982.744} C_VEL
LIN {X 0,Y 90.532,Z 939.048,A -85,B 0,C 180,E1 4969.349,E2 4969.349} C_VEL
LIN {X 0,Y 90.763,Z 940.997,A -85,B 0,C 180,E1 4956.96,E2 4956.96} C_VEL
LIN {X 0,Y 91.884,Z 941.432,A -85,B 0,C 180,E1 4950,E2 4950} C_VEL
LIN {X 0,Y 90.836,Z 940.851,A -85,B 0,C 180,E1 4941.772,E2 4941.772} C_VEL
LIN {X 0,Y 91.414,Z 938.653,A -85,B 0,C 180,E1 4928.841,E2 4928.841} C_VEL
LIN {X 0,Y 96.614,Z 934.465,A -85,B 0,C 180,E1 4915.304,E2 4915.304} C_VEL
LIN {X 0,Y 106.466,Z 928.428,A -85,B 0,C 180,E1 4903.683,E2 4903.683} C_VEL
LIN {X 0,Y 115.043,Z 923.428,A -85,B 0,C 180,E1 4897.31,E2 4897.31} C_VEL
LIN {X 0,Y 98.283,Z 917.708,A -85,B 0,C 180,E1 4878.384,E2 4878.384} C_VEL
LIN {X 0,Y 95.574,Z 911.594,A -85,B 0,C 180,E1 4853.392,E2 4853.392} C_VEL
LIN {X 0,Y 120.481,Z 902.974,A -85,B 0,C 180,E1 4823.306,E2 4823.306} C_VEL
LIN {X 0,Y 126.523,Z 901.616,A -85,B 0,C 180,E1 4820.048,E2 4820.048} C_VEL
LIN {X 0,Y 113.258,Z 908.513,A -85,B 0,C 180,E1 4811.463,E2 4811.463} C_VEL
LIN {X 0,Y 102.737,Z 913.467,A -85,B 0,C 180,E1 4801.053,E2 4801.053} C_VEL
LIN {X 0,Y 95.637,Z 916.618,A -85,B 0,C 180,E1 4788.912,E2 4788.912} C_VEL
LIN {X 0,Y 92.398,Z 918.07,A -85,B 0,C 180,E1 4776.213,E2 4776.213} C_VEL
LIN {X 0,Y 92.317,Z 918.094,A -85,B 0,C 180,E1 4764.406,E2 4764.406} C_VEL
LIN {X 0,Y 95.148,Z 916.84,A -85,B 0,C 180,E1 4752.257,E2 4752.257} C_VEL
LIN {X 0,Y 101.501,Z 914.044,A -85,B 0,C 180,E1 4740.492,E2 4740.492} C_VEL
LIN {X 0,Y 111.054,Z 909.628,A -85,B 0,C 180,E1 4730.264,E2 4730.264} C_VEL
LIN {X 0,Y 123.245,Z 903.471,A -85,B 0,C 180,E1 4721.703,E2 4721.703} C_VEL
LIN {X 0,Y 136.712,Z 895.88,A -85,B 0,C 180,E1 4715,E2 4715} C_VEL
LIN {X 0,Y 150.811,Z 886.928,A -85,B 0,C 180,E1 4709.711,E2 4709.711} C_VEL
LIN {X 0,Y 165.299,Z 876.511,A -85,B 0,C 180,E1 4705.435,E2 4705.435} C_VEL
LIN {X 0,Y 179.131,Z 865.234,A -85,B 0,C 180,E1 4702.091,E2 4702.091} C_VEL
LIN {X 0,Y 192.812,Z 852.576,A -85,B 0,C 180,E1 4699.297,E2 4699.297} C_VEL
LIN {X 0,Y 205.944,Z 838.715,A -85,B 0,C 180,E1 4696.969,E2 4696.969} C_VEL
LIN {X 0,Y 218.425,Z 823.602,A -85,B 0,C 180,E1 4695.006,E2 4695.006} C_VEL
LIN {X 0,Y 229.719,Z 807.819,A -85,B 0,C 180,E1 4693.389,E2 4693.389} C_VEL
LIN {X 0,Y 239.896,Z 791.267,A -85,B 0,C 180,E1 4692.029,E2 4692.029} C_VEL
LIN {X 0,Y 248.796,Z 774.223,A -85,B 0,C 180,E1 4690.888,E2 4690.888} C_VEL
LIN {X 0,Y 256.326,Z 757.022,A -85,B 0,C 180,E1 4689.948,E2 4689.948} C_VEL
LIN {X 0,Y 263.199,Z 737.453,A -85,B 0,C 180,E1 4689.069,E2 4689.069} C_VEL
LIN {X 0,Y 273.439,Z 703.168,A -85,B 0,C 180,E1 4687.851,E2 4687.851} C_VEL
LIN {X 0,Y 282.636,Z 668.648,A -85,B 0,C 180,E1 4686.945,E2 4686.945} C_VEL
LIN {X 0,Y 291.108,Z 631.644,A -85,B 0,C 180,E1 4686.256,E2 4686.256} C_VEL
LIN {X 0,Y 298.841,Z 589.7,A -85,B 0,C 180,E1 4685.651,E2 4685.651} C_VEL
LIN {X 0,Y 304.708,Z 547.493,A -85,B 0,C 180,E1 4685.109,E2 4685.109} C_VEL
LIN {X 0,Y 307.943,Z 520.078,A -85,B 0,C 180,E1 4684.749,E2 4684.749} C_VEL
LIN {X 0,Y 307.644,Z 517.482,A -85,B 0,C 180,E1 4682.422,E2 4682.422} C_VEL
LIN {X 0,Y 307.613,Z 517.161,A -85,B 0,C 180,E1 4681.882,E2 4681.882} C_VEL
LIN {X 0,Y 299.156,Z 582.532,A -85,B 0,C 180,E1 4680.849,E2 4680.849} C_VEL
LIN {X 0,Y 292.355,Z 622.413,A -85,B 0,C 180,E1 4680.235,E2 4680.235} C_VEL
LIN {X 0,Y 283.768,Z 662.379,A -85,B 0,C 180,E1 4679.639,E2 4679.639} C_VEL
LIN {X 0,Y 273.179,Z 702.835,A -85,B 0,C 180,E1 4678.87,E2 4678.87} C_VEL
LIN {X 0,Y 261.634,Z 740.122,A -85,B 0,C 180,E1 4677.975,E2 4677.975} C_VEL
LIN {X 0,Y 252.78,Z 765.045,A -85,B 0,C 180,E1 4677.169,E2 4677.169} C_VEL
LIN {X 0,Y 248.861,Z 774.442,A -85,B 0,C 180,E1 4676.794,E2 4676.794} C_VEL
LIN {X 0,Y 245.415,Z 781.761,A -85,B 0,C 180,E1 4676.711,E2 4676.711} C_VEL
LIN {X 0,Y 235.59,Z 799.084,A -85,B 0,C 180,E1 4677.307,E2 4677.307} C_VEL
LIN {X 0,Y 231.635,Z 805.444,A -85,B 0,C 180,E1 4677.201,E2 4677.201} C_VEL
LIN {X 0,Y 220.49,Z 822.504,A -85,B 0,C 180,E1 4676.086,E2 4676.086} C_VEL
LIN {X 0,Y 208.44,Z 838.497,A -85,B 0,C 180,E1 4674.771,E2 4674.771} C_VEL
LIN {X 0,Y 194.433,Z 854.698,A -85,B 0,C 180,E1 4672.986,E2 4672.986} C_VEL
LIN {X 0,Y 179.35,Z 869.944,A -85,B 0,C 180,E1 4670.676,E2 4670.676} C_VEL
LIN {X 0,Y 163.704,Z 883.811,A -85,B 0,C 180,E1 4667.759,E2 4667.759} C_VEL
LIN {X 0,Y 147.139,Z 896.754,A -85,B 0,C 180,E1 4663.822,E2 4663.822} C_VEL
LIN {X 0,Y 130.928,Z 908.015,A -85,B 0,C 180,E1 4658.702,E2 4658.702} C_VEL
LIN {X 0,Y 115.543,Z 917.657,A -85,B 0,C 180,E1 4651.968,E2 4651.968} C_VEL
LIN {X 0,Y 101.578,Z 925.785,A -85,B 0,C 180,E1 4642.875,E2 4642.875} C_VEL
LIN {X 0,Y 90.768,Z 932.047,A -85,B 0,C 180,E1 4631.372,E2 4631.372} C_VEL
LIN {X 0,Y 84.153,Z 936.564,A -85,B 0,C 180,E1 4617.606,E2 4617.606} C_VEL
LIN {X 0,Y 82.324,Z 939.385,A -85,B 0,C 180,E1 4602.628,E2 4602.628} C_VEL
LIN {X 0,Y 83.705,Z 940.369,A -85,B 0,C 180,E1 4591.369,E2 4591.369} C_VEL
LIN {X 0,Y 83.795,Z 940.376,A -85,B 0,C 180,E1 4588.632,E2 4588.632} C_VEL
LIN {X 0,Y 82.683,Z 939.337,A -85,B 0,C 180,E1 4576.716,E2 4576.716} C_VEL
LIN {X 0,Y 85.426,Z 936.323,A -85,B 0,C 180,E1 4561.321,E2 4561.321} C_VEL
LIN {X 0,Y 93.941,Z 931.168,A -85,B 0,C 180,E1 4547.061,E2 4547.061} C_VEL
LIN {X 0,Y 105.206,Z 924.983,A -85,B 0,C 180,E1 4536.951,E2 4536.951} C_VEL
LIN {X 0,Y 87.962,Z 914.352,A -85,B 0,C 180,E1 4493.473,E2 4493.473} C_VEL
LIN {X 0,Y 113.972,Z 905.824,A -85,B 0,C 180,E1 4461.335,E2 4461.335} C_VEL
LIN {X 0,Y 116.137,Z 905.376,A -85,B 0,C 180,E1 4460.019,E2 4460.019} C_VEL
LIN {X 0,Y 102.89,Z 911.534,A -85,B 0,C 180,E1 4450.626,E2 4450.626} C_VEL
LIN {X 0,Y 92.681,Z 915.818,A -85,B 0,C 180,E1 4439.044,E2 4439.044} C_VEL
LIN {X 0,Y 86.506,Z 918.256,A -85,B 0,C 180,E1 4426.106,E2 4426.106} C_VEL
LIN {X 0,Y 84.155,Z 919.174,A -85,B 0,C 180,E1 4412.725,E2 4412.725} C_VEL
LIN {X 0,Y 85.139,Z 918.795,A -85,B 0,C 180,E1 4399.17,E2 4399.17} C_VEL
LIN {X 0,Y 89.844,Z 916.965,A -85,B 0,C 180,E1 4385.684,E2 4385.684} C_VEL
LIN {X 0,Y 98.736,Z 913.368,A -85,B 0,C 180,E1 4373.31,E2 4373.31} C_VEL
LIN {X 0,Y 110.955,Z 907.949,A -85,B 0,C 180,E1 4363.119,E2 4363.119} C_VEL
LIN {X 0,Y 124.281,Z 901.313,A -85,B 0,C 180,E1 4355.651,E2 4355.651} C_VEL
LIN {X 0,Y 138.369,Z 893.378,A -85,B 0,C 180,E1 4349.872,E2 4349.872} C_VEL
LIN {X 0,Y 153.498,Z 883.669,A -85,B 0,C 180,E1 4345.117,E2 4345.117} C_VEL
LIN {X 0,Y 168.553,Z 872.614,A -85,B 0,C 180,E1 4341.353,E2 4341.353} C_VEL
LIN {X 0,Y 183.271,Z 860.256,A -85,B 0,C 180,E1 4338.321,E2 4338.321} C_VEL
LIN {X 0,Y 197.009,Z 847.042,A -85,B 0,C 180,E1 4335.907,E2 4335.907} C_VEL
LIN {X 0,Y 210.573,Z 832.06,A -85,B 0,C 180,E1 4333.82,E2 4333.82} C_VEL
LIN {X 0,Y 222.939,Z 816.241,A -85,B 0,C 180,E1 4332.113,E2 4332.113} C_VEL
LIN {X 0,Y 234.043,Z 799.685,A -85,B 0,C 180,E1 4330.698,E2 4330.698} C_VEL
LIN {X 0,Y 244.295,Z 781.633,A -85,B 0,C 180,E1 4329.459,E2 4329.459} C_VEL
LIN {X 0,Y 252.728,Z 763.766,A -85,B 0,C 180,E1 4328.469,E2 4328.469} C_VEL
LIN {X 0,Y 260.245,Z 744.124,A -85,B 0,C 180,E1 4327.579,E2 4327.579} C_VEL
LIN {X 0,Y 270.884,Z 710.049,A -85,B 0,C 180,E1 4326.373,E2 4326.373} C_VEL
LIN {X 0,Y 280.975,Z 673.445,A -85,B 0,C 180,E1 4325.419,E2 4325.419} C_VEL
LIN {X 0,Y 289.674,Z 636.145,A -85,B 0,C 180,E1 4324.745,E2 4324.745} C_VEL
LIN {X 0,Y 297.291,Z 596.179,A -85,B 0,C 180,E1 4324.2,E2 4324.2} C_VEL
LIN {X 0,Y 303.116,Z 556.268,A -85,B 0,C 180,E1 4323.707,E2 4323.707} C_VEL
LIN {X 0,Y 306.729,Z 526.374,A -85,B 0,C 180,E1 4323.317,E2 4323.317} C_VEL
LIN {X 0,Y 306.69,Z 526.528,A -85,B 0,C 180,E1 4323.235,E2 4323.235} C_VEL
LIN {X 0,Y 299.195,Z 582.451,A -85,B 0,C 180,E1 4322.387,E2 4322.387} C_VEL
LIN {X 0,Y 292.364,Z 621.539,A -85,B 0,C 180,E1 4321.816,E2 4321.816} C_VEL
LIN {X 0,Y 283.917,Z 660.513,A -85,B 0,C 180,E1 4321.287,E2 4321.287} C_VEL
LIN {X 0,Y 273.328,Z 700.792,A -85,B 0,C 180,E1 4320.591,E2 4320.591} C_VEL
LIN {X 0,Y 261.972,Z 737.428,A -85,B 0,C 180,E1 4319.802,E2 4319.802} C_VEL
LIN {X 0,Y 253.005,Z 762.644,A -85,B 0,C 180,E1 4319.071,E2 4319.071} C_VEL
LIN {X 0,Y 244.576,Z 781.78,A -85,B 0,C 180,E1 4318.341,E2 4318.341} C_VEL
LIN {X 0,Y 234.209,Z 801.18,A -85,B 0,C 180,E1 4317.433,E2 4317.433} C_VEL
LIN {X 0,Y 231.635,Z 805.444,A -85,B 0,C 180,E1 4317.201,E2 4317.201} C_VEL
LIN {X 0,Y 227.509,Z 812.018,A -85,B 0,C 180,E1 4317.07,E2 4317.07} C_VEL
LIN {X 0,Y 215.453,Z 828.05,A -85,B 0,C 180,E1 4317.542,E2 4317.542} C_VEL
LIN {X 0,Y 210.544,Z 834.012,A -85,B 0,C 180,E1 4317.339,E2 4317.339} C_VEL
LIN {X 0,Y 196.509,Z 850.413,A -85,B 0,C 180,E1 4315.787,E2 4315.787} C_VEL
LIN {X 0,Y 182.009,Z 865.202,A -85,B 0,C 180,E1 4313.903,E2 4313.903} C_VEL
LIN {X 0,Y 165.684,Z 879.722,A -85,B 0,C 180,E1 4311.322,E2 4311.322} C_VEL
LIN {X 0,Y 149.238,Z 892.561,A -85,B 0,C 180,E1 4308.012,E2 4308.012} C_VEL
LIN {X 0,Y 132.381,Z 904.133,A -85,B 0,C 180,E1 4303.585,E2 4303.585} C_VEL
LIN {X 0,Y 114.956,Z 914.714,A -85,B 0,C 180,E1 4297.219,E2 4297.219} C_VEL
LIN {X 0,Y 99.405,Z 923.251,A -85,B 0,C 180,E1 4288.758,E2 4288.758} C_VEL
LIN {X 0,Y 86.671,Z 929.904,A -85,B 0,C 180,E1 4277.59,E2 4277.59} C_VEL
LIN {X 0,Y 77.683,Z 934.991,A -85,B 0,C 180,E1 4262.724,E2 4262.724} C_VEL
LIN {X 0,Y 74.38,Z 938.082,A -85,B 0,C 180,E1 4246.397,E2 4246.397} C_VEL
LIN {X 0,Y 75.401,Z 939.275,A -85,B 0,C 180,E1 4233.04,E2 4233.04} C_VEL
LIN {X 0,Y 75.898,Z 939.4,A -85,B 0,C 180,E1 4229.245,E2 4229.245} C_VEL
LIN {X 0,Y 74.73,Z 938.387,A -85,B 0,C 180,E1 4216.063,E2 4216.063} C_VEL
LIN {X 0,Y 78.008,Z 935.438,A -85,B 0,C 180,E1 4199.155,E2 4199.155} C_VEL
LIN {X 0,Y 87.07,Z 930.614,A -85,B 0,C 180,E1 4184.468,E2 4184.468} C_VEL
LIN {X 0,Y 95.561,Z 926.36,A -85,B 0,C 180,E1 4176.613,E2 4176.613} C_VEL
LIN {X 0,Y 80.507,Z 916.643,A -85,B 0,C 180,E1 4132.148,E2 4132.148} C_VEL
LIN {X 0,Y 105.806,Z 908.837,A -85,B 0,C 180,E1 4100.059,E2 4100.059} C_VEL
LIN {X 0,Y 92.509,Z 914.309,A -85,B 0,C 180,E1 4089.622,E2 4089.622} C_VEL
LIN {X 0,Y 82.543,Z 917.978,A -85,B 0,C 180,E1 4076.31,E2 4076.31} C_VEL
LIN {X 0,Y 77.216,Z 919.83,A -85,B 0,C 180,E1 4061.201,E2 4061.201} C_VEL
LIN {X 0,Y 76.265,Z 920.164,A -85,B 0,C 180,E1 4046.242,E2 4046.242} C_VEL
LIN {X 0,Y 79.269,Z 919.146,A -85,B 0,C 180,E1 4031.094,E2 4031.094} C_VEL
LIN {X 0,Y 86.613,Z 916.566,A -85,B 0,C 180,E1 4017.141,E2 4017.141} C_VEL
LIN {X 0,Y 97.498,Z 912.41,A -85,B 0,C 180,E1 4005.784,E2 4005.784} C_VEL
LIN {X 0,Y 111.108,Z 906.536,A -85,B 0,C 180,E1 3996.781,E2 3996.781} C_VEL
LIN {X 0,Y 125.894,Z 899.224,A -85,B 0,C 180,E1 3990.025,E2 3990.025} C_VEL
LIN {X 0,Y 141.089,Z 890.591,A -85,B 0,C 180,E1 3984.889,E2 3984.889} C_VEL
LIN {X 0,Y 156.263,Z 880.695,A -85,B 0,C 180,E1 3980.899,E2 3980.899} C_VEL
LIN {X 0,Y 171.564,Z 869.227,A -85,B 0,C 180,E1 3977.642,E2 3977.642} C_VEL
LIN {X 0,Y 185.439,Z 857.363,A -85,B 0,C 180,E1 3975.167,E2 3975.167} C_VEL
LIN {X 0,Y 199.581,Z 843.46,A -85,B 0,C 180,E1 3972.984,E2 3972.984} C_VEL
LIN {X 0,Y 212.537,Z 828.799,A -85,B 0,C 180,E1 3971.217,E2 3971.217} C_VEL
LIN {X 0,Y 224.695,Z 812.848,A -85,B 0,C 180,E1 3969.711,E2 3969.711} C_VEL
LIN {X 0,Y 235.537,Z 796.244,A -85,B 0,C 180,E1 3968.46,E2 3968.46} C_VEL
LIN {X 0,Y 245.494,Z 778.148,A -85,B 0,C 180,E1 3967.357,E2 3967.357} C_VEL
LIN {X 0,Y 254.068,Z 759.222,A -85,B 0,C 180,E1 3966.426,E2 3966.426} C_VEL
LIN {X 0,Y 261.948,Z 737.318,A -85,B 0,C 180,E1 3965.549,E2 3965.549} C_VEL
LIN {X 0,Y 272.925,Z 701.674,A -85,B 0,C 180,E1 3964.436,E2 3964.436} C_VEL
LIN {X 0,Y 282.567,Z 665.721,A -85,B 0,C 180,E1 3963.632,E2 3963.632} C_VEL
LIN {X 0,Y 288.838,Z 638.838,A -85,B 0,C 180,E1 3963.188,E2 3963.188} C_VEL
LIN {X 0,Y 279.381,Z 678.226,A -85,B 0,C 180,E1 3962.643,E2 3962.643} C_VEL
LIN {X 0,Y 267.773,Z 718.617,A -85,B 0,C 180,E1 3961.95,E2 3961.95} C_VEL
LIN {X 0,Y 256.526,Z 752.173,A -85,B 0,C 180,E1 3961.181,E2 3961.181} C_VEL
LIN {X 0,Y 248.987,Z 770.899,A -85,B 0,C 180,E1 3960.622,E2 3960.622} C_VEL
LIN {X 0,Y 239.61,Z 789.996,A -85,B 0,C 180,E1 3959.891,E2 3959.891} C_VEL
LIN {X 0,Y 229.006,Z 808.108,A -85,B 0,C 180,E1 3959.044,E2 3959.044} C_VEL
